ABB RAPID module: TaskModule.mod

MODULE TaskModule
    !*****************************************************
    !Module Name: TaskModule
    !Version:     1.0
    !Description: This module stroes ths data which are not shared among other tasks
    !Date:        2018-8-10
    !Author:      Michael
    !*****************************************************

    VAR num numStation:=1;
    VAR partdata pdTmpChk;
    VAR string sPartDataName;

    VAR syncident SyncPositionerHomed;
    VAR syncident SyncWobjScanning;
    VAR syncident SyncWobjBranchScaning;
    VAR syncident SyncWobjBranchScaned;
    VAR syncident SyncWobjHeaderScaning;
    VAR syncident SyncWobjHeaderScaned;
    VAR syncident SyncWobjBranchScaningV2;
    VAR syncident SyncWobjBranchScanedV2;
    VAR syncident SyncWobjHeaderScaningV2;
    VAR syncident SyncWobjHeaderScanedV2;
    VAR syncident SyncBranchPeripherySmarTac;
    VAR syncident SyncHeaderPeripherySmarTac;
    VAR syncident SyncWobjScaned;
    VAR syncident SyncWobjRevised;

    VAR syncident SyncPositionerWeldApproached;
    VAR syncident SyncRobotsWeldApproached;
    VAR syncident SyncAllRobotsWeldStart;
    VAR syncident SyncAllRobotsWeldEnd;
    VAR syncident SyncRobotsWeldDeparted;

    VAR syncident SyncMoveLSubstituted1;
    VAR syncident SyncMoveLSubstituted2;

    VAR syncident SyncRobotsForTest11;
    VAR syncident SyncRobotsForTest12;
    VAR syncident SyncRobotsForTest13;

    VAR syncident SyncRobotsForTest21;
    VAR syncident SyncRobotsForTest22;
    VAR syncident SyncRobotsForTest23;
    VAR syncident SyncRobotsForTest24;
    VAR syncident SyncRobotsForTest25;
    VAR syncident SyncRobotsForTest26;

    VAR syncident SyncVerifyTrackHorizontal1;
    VAR syncident SyncVerifyTrackHorizontal2;
    VAR syncident SyncVerifyTrackHorizontal3;
    VAR syncident SyncVerifyTrackHorizontal4;
    VAR syncident SyncVerifyTrackHorizontal5;
    VAR syncident SyncVerifyTrackHorizontal6;
    VAR syncident SyncVerifyTrackHorizontal7;
    VAR syncident SyncVerifyTrackHorizontal8;

    VAR string strCurTaskName:="T_ROB2";
    VAR num numCurTaskNo:=2;
    VAR num numRobLayerCurTotal;
    VAR RECORDWeldTarget rRobLayerCur{30};

    TASK PERS tooldata toolWeldGun:=[TRUE,[[79.6797,-0.416093,372.923],[0.951182,0.000468257,0.308629,0.000774227]],[5.2,[30.6,-22.1,100.1],[1,0,0,0],0,0,0]];
    TASK PERS tooldata toolLaser:=[TRUE,[[-50.2332,13.2462,422.412],[0.99997,-0.00371251,-0.00510598,-0.00440267]],[5.2,[30.6,-22.1,100.1],[1,0,0,0],0,0,0]];
    TASK PERS extjoint extjointValue:=[3962.74,9E+09,9E+09,9E+09,9E+09,9E+09];

    TASK PERS robtarget robtApproachPlatoonSinking:=[[380,200,190.09],[0.24541,0.749,0.614742,-0.0294245],[-1,-1,0,1],[4837,9E+09,9E+09,9E+09,9E+09,9E+09]];
    TASK PERS robtarget robtDepartPlatoonSinking:=[[380,200,190.09],[0.245412,0.748999,0.614742,-0.0294268],[-1,-1,0,1],[4837,9E+09,9E+09,9E+09,9E+09,9E+09]];

    TASK PERS robtarget robtApproachSaddle:=[[487.15,620.91,295.61],[0.42303,-0.434139,-0.767759,0.207644],[0,-1,0,0],[4837,9E+09,9E+09,9E+09,9E+09,9E+09]];
    TASK PERS robtarget robtDepartSaddle:=[[487.15,238.1,333.7],[0.270598,0.653282,-0.653281,0.270598],[0,-1,-2,0],[4837,9E+09,9E+09,9E+09,9E+09,9E+09]];

    TASK PERS robtarget robtApproachSaddleScan:=[[380,426.46,263.71],[0.0219383,0.0029599,-0.868719,0.494811],[-1,-1,-1,1],[4837,9E+09,9E+09,9E+09,9E+09,9E+09]];
    TASK PERS robtarget robtDepartSaddleScan:=[[380,426.46,263.71],[0.0219385,0.00296103,-0.868717,0.494814],[-1,-1,-1,1],[4837,9E+09,9E+09,9E+09,9E+09,9E+09]];

    TASK PERS robtarget robtApproachPlatoonSinkingScan:=[[380,238.1,333.7],[0.270598,0.653281,-0.653282,0.270598],[0,0,1,1],[4837,9E+09,9E+09,9E+09,9E+09,9E+09]];
    TASK PERS robtarget robtDepartPlatoonSinkingScan:=[[380,238.1,333.7],[0.270598,0.653281,-0.653282,0.270598],[0,0,1,1],[4837,9E+09,9E+09,9E+09,9E+09,9E+09]];

    TASK PERS confdata confPlatoonSinkingOrigin:=[0,0,0,1];
    TASK PERS confdata confSaddleOrigin:=[0,-1,0,0];

    TASK PERS robtarget robtNext:=[[39.1752,-5.3,137.55],[0.0379422,0.543848,0.68392,-0.484813],[0,0,-1,1],[447,9E+09,9E+09,9E+09,9E+09,9E+09]];
    TASK PERS robtarget robtCircleEnd:=[[37.5661,-7.30249,138.697],[0.0379422,0.543848,0.68392,-0.484813],[-1,-1,-1,1],[2602,9E+09,9E+09,9E+09,9E+09,9E+09]];

    TASK PERS seamdata seamNext:=[0,0.5,[0,0,0,100,0,0,0,0,0],0,0,5,0,0,[0,0,1,140,0,0,0,0,0],0,1.5,[0,0,1,90,0,0,0,0,0],0.04,0,[0,0,0,0,0,0,0,0,0],0.5];
    TASK PERS welddata weldNext:=[7,0,[25,0,0,0,0,200,0,0,0],[0,0,0,0,0,0,0,0,0]];
    TASK PERS weavedata weaveNext:=[0,0,0,0,0,0,0,0,0,0,0,0,0,0,0];
    TASK PERS trackdata trackNext:=[0,FALSE,50,[0,0,0,0,0,0,0,0,0],[0,0,0,0,0,0,0]];
    TASK PERS adaptdata adaptNext:=[0,1,0,0,0.1,100,0.1,100];
    TASK PERS num numWeaveWidth90:=0;
    TASK PERS num numGrooveWidthNext:=0.1;

    TASK PERS jointtarget jointNext:=[[9E+09,9E+09,9E+09,9E+09,9E+09,9E+09],[0,66.4272,9E+09,9E+09,9E+09,9E+09]];

    VAR clock clockPartTimeConsume;
    TASK PERS num numTimeConsumeTotal:=683.013;

    CONST string strWeldProcedureLogLogFileName:="WeldProcedureLog2.csv";

    CONST string strSSBLogFileName:="ScanSaddleBranch2.csv";
    CONST string strSSHLogFileName:="ScanSaddleHeader2.csv";

    !For branch SmarTac
    TASK PERS num numSSBPointsTotal:=13;
    !Scan branch range
    TASK PERS num numSSBAngleFrom:=125;
    TASK PERS num numSSBAngleTo:=30;

    !For saddle header SmarTac
    TASK PERS num numSSHPointsTotal:=13;
    !Scan saddle header range
    TASK PERS num numSSHAngleFrom:=0;
    TASK PERS num numSSHAngleTo:=90;

    !Scan saddle branch points
    TASK PERS robtarget robtSSBLaserSmarTacs{20}:=[[[923.658,130.45,259.25],[0.67438,0.67438,0.212631,0.212631],[-1,-1,1,1],[4202,9E+09,9E+09,9E+09,9E+09,9E+09]],[[942.496,141.787,259.25],[0.687449,0.687449,0.165571,0.165571],[-1,-1,1,1],[4202,9E+09,9E+09,9E+09,9E+09,9E+09]],[[962.716,150.422,259.25],[0.697239,0.697239,0.11772,0.11772],[-1,-1,1,1],[4202,9E+09,9E+09,9E+09,9E+09,9E+09]],[[983.932,156.19,259.25],[0.703702,0.703702,0.0693086,0.0693086],[-1,-1,1,1],[4202,9E+09,9E+09,9E+09,9E+09,9E+09]],[[1005.74,158.981,259.25],[0.706808,0.706808,0.020566,0.020566],[-1,-1,1,1],[4202,9E+09,9E+09,9E+09,9E+09,9E+09]],[[1027.73,158.741,259.25],[0.706541,0.706541,-0.0282747,-0.0282747],[0,0,1,1],[4202,9E+09,9E+09,9E+09,9E+09,9E+09]],[[1049.47,155.475,259.25],[0.702904,0.702904,-0.0769805,-0.0769805],[0,0,0,1],[4202,9E+09,9E+09,9E+09,9E+09,9E+09]],[[1070.55,149.246,259.25],[0.695913,0.695913,-0.125319,-0.125319],[0,0,0,1],[4202,9E+09,9E+09,9E+09,9E+09,9E+09]],[[1090.58,140.172,259.25],[0.685602,0.685602,-0.17306,-0.17306],[0,0,0,1],[4202,9E+09,9E+09,9E+09,9E+09,9E+09]],[[1109.17,128.426,259.25],[0.67202,0.67202,-0.219975,-0.219975],[0,0,0,1],[4202,9E+09,9E+09,9E+09,9E+09,9E+09]],[[1125.96,114.233,259.25],[0.655232,0.655232,-0.26584,-0.26584],[0,0,0,1],[4202,9E+09,9E+09,9E+09,9E+09,9E+09]],[[1140.63,97.8615,259.25],[0.635318,0.635318,-0.310437,-0.310437],[0,0,0,1],[4202,9E+09,9E+09,9E+09,9E+09,9E+09]],[[1152.91,79.625,259.25],[0.612372,0.612372,-0.353553,-0.353553],[0,0,0,1],[4202,9E+09,9E+09,9E+09,9E+09,9E+09]],[[652.53,-493.33,1047.99],[0.459259,-0.544323,-0.447932,-0.54051],[0,0,0,1],[4837,9E+09,9E+09,9E+09,9E+09,9E+09]],[[652.53,-493.33,1047.99],[0.459259,-0.544323,-0.447932,-0.54051],[-1,0,-2,1],[4837,9E+09,9E+09,9E+09,9E+09,9E+09]],[[652.53,-493.33,1047.99],[0.459259,-0.544323,-0.447932,-0.54051],[-1,0,-2,1],[4837,9E+09,9E+09,9E+09,9E+09,9E+09]],[[652.53,-493.33,1047.99],[0.459259,-0.544323,-0.447932,-0.54051],[-1,0,-2,1],[4837,9E+09,9E+09,9E+09,9E+09,9E+09]],[[652.53,-493.33,1047.99],[0.459259,-0.544323,-0.447932,-0.54051],[-1,0,-2,1],[4837,9E+09,9E+09,9E+09,9E+09,9E+09]],[[652.53,-493.33,1047.99],[0.459259,-0.544323,-0.447932,-0.54051],[-1,0,-2,1],[4837,9E+09,9E+09,9E+09,9E+09,9E+09]],[[652.53,-493.33,1047.99],[0.459259,-0.544323,-0.447932,-0.54051],[-1,0,-2,1],[4837,9E+09,9E+09,9E+09,9E+09,9E+09]]];
    TASK PERS robtarget robtSSBWireSmarTacs{20}:=[[[428.493,28.575,188.15],[0.683013,0.183013,-0.683013,0.183013],[0,1,-3,1],[4838,9E+09,9E+09,9E+09,9E+09,9E+09]],[[422.779,36.7353,188.15],[0.664463,0.241845,-0.664463,0.241845],[0,1,-3,1],[4838,9E+09,9E+09,9E+09,9E+09,9E+09]],[[415.735,43.7794,188.15],[0.640856,0.298836,-0.640856,0.298836],[0,1,-3,1],[4838,9E+09,9E+09,9E+09,9E+09,9E+09]],[[407.575,49.4934,188.15],[0.612372,0.353553,-0.612372,0.353553],[0,0,-3,1],[4838,9E+09,9E+09,9E+09,9E+09,9E+09]],[[398.546,53.7034,188.15],[0.579228,0.40558,-0.579228,0.40558],[0,0,-3,1],[4838,9E+09,9E+09,9E+09,9E+09,9E+09]],[[388.924,56.2818,188.15],[0.541675,0.454519,-0.541675,0.454519],[0,0,-3,1],[4838,9E+09,9E+09,9E+09,9E+09,9E+09]],[[379,57.15,188.15],[0.5,0.5,-0.5,0.5],[0,0,-3,1],[4838,9E+09,9E+09,9E+09,9E+09,9E+09]],[[369.076,56.2818,188.15],[0.454519,0.541675,-0.454519,0.541675],[-1,-1,-2,1],[4838,9E+09,9E+09,9E+09,9E+09,9E+09]],[[359.454,53.7034,188.15],[0.40558,0.579228,-0.40558,0.579228],[-1,-1,-2,1],[4838,9E+09,9E+09,9E+09,9E+09,9E+09]],[[350.425,49.4934,188.15],[0.353553,0.612372,-0.353553,0.612372],[-1,-1,-2,1],[4838,9E+09,9E+09,9E+09,9E+09,9E+09]],[[342.265,43.7794,188.15],[0.298836,0.640856,-0.298836,0.640856],[-1,-2,-2,1],[4838,9E+09,9E+09,9E+09,9E+09,9E+09]],[[335.221,36.7353,188.15],[0.241845,0.664463,-0.241845,0.664463],[-1,-2,-2,1],[4838,9E+09,9E+09,9E+09,9E+09,9E+09]],[[329.507,28.575,188.15],[0.183013,0.683013,-0.183013,0.683013],[-1,-2,-2,1],[4838,9E+09,9E+09,9E+09,9E+09,9E+09]],[[652.53,-493.33,1047.99],[0.459259,-0.544323,-0.447932,-0.54051],[-1,-1,-2,1],[4837,9E+09,9E+09,9E+09,9E+09,9E+09]],[[652.53,-493.33,1047.99],[0.459259,-0.544323,-0.447932,-0.54051],[-1,0,-2,1],[4837,9E+09,9E+09,9E+09,9E+09,9E+09]],[[652.53,-493.33,1047.99],[0.459259,-0.544323,-0.447932,-0.54051],[-1,0,-2,1],[4837,9E+09,9E+09,9E+09,9E+09,9E+09]],[[652.53,-493.33,1047.99],[0.459259,-0.544323,-0.447932,-0.54051],[-1,0,-2,1],[4837,9E+09,9E+09,9E+09,9E+09,9E+09]],[[652.53,-493.33,1047.99],[0.459259,-0.544323,-0.447932,-0.54051],[-1,0,-2,1],[4837,9E+09,9E+09,9E+09,9E+09,9E+09]],[[652.53,-493.33,1047.99],[0.459259,-0.544323,-0.447932,-0.54051],[-1,0,-2,1],[4837,9E+09,9E+09,9E+09,9E+09,9E+09]],[[652.53,-493.33,1047.99],[0.459259,-0.544323,-0.447932,-0.54051],[-1,0,-2,1],[4837,9E+09,9E+09,9E+09,9E+09,9E+09]]];
    TASK PERS robtarget robtSSBLinerFrom:=[[427.815,90,259.25],[0.707107,0.707107,0,0],[0,0,1,1],[4202,9E+09,9E+09,9E+09,9E+09,9E+09]];
    TASK PERS robtarget robtSSBLinerTo:=[[427.815,90,259.25],[0.707107,0.707107,0,0],[0,0,1,1],[4202,9E+09,9E+09,9E+09,9E+09,9E+09]];

    !Scan saddle branch results, shared for all the four scan methods
    TASK PERS pose poseSSBs{20}:=[[[-1.32358,1.90598,0.00161743],[1,0,0,0]],[[-0.951538,1.84398,-0.0424805],[1,0,0,0]],[[-0.775452,2.22177,-0.0251465],[1,0,0,0]],[[-0.413208,2.22758,0.000427246],[1,0,0,0]],[[-0.156219,2.60087,-0.0246429],[1,0,0,0]],[[0.213074,2.58353,0.020462],[1,0,0,0]],[[0.449005,2.08419,-0.0298309],[1,0,0,0]],[[0.743073,1.96958,-0.0420227],[1,0,0,0]],[[1.15472,2.18119,0.0494232],[1,0,0,0]],[[1.04321,1.4268,-0.00532532],[1,0,0,0]],[[1.86594,1.89365,0.0466766],[1,0,0,0]],[[1.22217,0.918324,-0.00390625],[1,0,0,0]],[[0.608215,0.37476,-0.00968933],[1,0,0,0]],[[0,0,0],[1,0,0,0]],[[0,0,0],[1,0,0,0]],[[0,0,0],[1,0,0,0]],[[0,0,0],[1,0,0,0]],[[0,0,0],[1,0,0,0]],[[0,0,0],[1,0,0,0]],[[0,0,0],[1,0,0,0]]];
    TASK PERS num numSSBLaserValues{100}:=[0,0,0,0,0,0,0,0,0,0,0,0,0,0,0,0,0,0,0,0,0,0,0,0,0,0,0,0,0,0,0,0,0,0,0,0,0,0,0,0,0,0,0,0,0,0,0,0,0,0,0,0,0,0,0,0,0,0,0,0,0,0,0,0,0,0,0,0,0,0,0,0,0,0,0,0,0,0,0,0,0,0,0,0,0,0,0,0,0,0,0,0,0,0,0,0,0,0,0,0];
    TASK PERS robtarget robtSSBPeripherys{100}:=[[[345.897,48.7205,208.152],[0.674376,0.674381,0.212635,0.212635],[-1,-1,1,1],[4837,9E+09,9E+09,9E+09,9E+09,9E+09]],[[353.029,52.7272,208.108],[0.687429,0.687473,0.165559,0.165568],[-1,-1,1,1],[4837,9E+09,9E+09,9E+09,9E+09,9E+09]],[[360.461,56.2038,208.125],[0.697234,0.697245,0.117717,0.11772],[-1,-1,1,1],[4837,9E+09,9E+09,9E+09,9E+09,9E+09]],[[368.437,58.2795,208.15],[0.703708,0.703694,0.0693283,0.0693077],[-1,-1,1,1],[4837,9E+09,9E+09,9E+09,9E+09,9E+09]],[[376.521,59.6542,208.125],[0.706794,0.706822,0.0205642,0.0205642],[-1,-1,1,1],[4837,9E+09,9E+09,9E+09,9E+09,9E+09]],[[384.78,59.5508,208.17],[0.706548,0.706534,-0.0282861,-0.0282663],[0,0,0,1],[4837,9E+09,9E+09,9E+09,9E+09,9E+09]],[[392.819,57.8795,208.12],[0.702889,0.702918,-0.0769979,-0.0769742],[0,0,0,1],[4836.99,9E+09,9E+09,9E+09,9E+09,9E+09]],[[400.68,55.5295,208.108],[0.695903,0.695926,-0.125326,-0.125296],[0,0,0,1],[4837,9E+09,9E+09,9E+09,9E+09,9E+09]],[[408.278,52.4847,208.199],[0.685623,0.685578,-0.173065,-0.173068],[0,0,0,1],[4837,9E+09,9E+09,9E+09,9E+09,9E+09]],[[414.837,47.5151,208.145],[0.672022,0.672019,-0.219953,-0.219993],[0,0,0,1],[4837,9E+09,9E+09,9E+09,9E+09,9E+09]],[[421.685,42.8883,208.197],[0.655247,0.655221,-0.265826,-0.265844],[0,0,0,1],[4837,9E+09,9E+09,9E+09,9E+09,9E+09]],[[426.308,36.0378,208.146],[0.635315,0.635323,-0.310461,-0.310408],[0,0,0,1],[4837,9E+09,9E+09,9E+09,9E+09,9E+09]],[[430.102,28.9498,208.14],[0.612373,0.612366,-0.353539,-0.353577],[0,0,0,1],[4837,9E+09,9E+09,9E+09,9E+09,9E+09]],[[75.54,-110.49,75.53],[0.104911,-0.592891,0.59209,0.535634],[-1,-2,0,1],[3747.5,9E+09,9E+09,9E+09,9E+09,9E+09]],[[75.54,-110.49,75.53],[0.104911,-0.592891,0.59209,0.535634],[-1,0,-1,0],[3747.5,9E+09,9E+09,9E+09,9E+09,9E+09]],[[75.54,-110.49,75.53],[0.104911,-0.592891,0.59209,0.535634],[-1,0,-1,0],[3747.5,9E+09,9E+09,9E+09,9E+09,9E+09]],[[75.54,-110.49,75.53],[0.104911,-0.592891,0.59209,0.535634],[-1,0,-1,0],[3747.5,9E+09,9E+09,9E+09,9E+09,9E+09]],[[75.54,-110.49,75.53],[0.104911,-0.592891,0.59209,0.535634],[-1,0,-1,0],[3747.5,9E+09,9E+09,9E+09,9E+09,9E+09]],[[75.54,-110.49,75.53],[0.104911,-0.592891,0.59209,0.535634],[-1,0,-1,0],[3747.5,9E+09,9E+09,9E+09,9E+09,9E+09]],[[75.54,-110.49,75.53],[0.104911,-0.592891,0.59209,0.535634],[-1,0,-1,0],[3747.5,9E+09,9E+09,9E+09,9E+09,9E+09]],[[75.54,-110.49,75.53],[0.104911,-0.592891,0.59209,0.535634],[-1,0,-1,0],[3747.5,9E+09,9E+09,9E+09,9E+09,9E+09]],[[75.54,-110.49,75.53],[0.104911,-0.592891,0.59209,0.535634],[-1,0,-1,0],[3747.5,9E+09,9E+09,9E+09,9E+09,9E+09]],[[75.54,-110.49,75.53],[0.104911,-0.592891,0.59209,0.535634],[-1,0,-1,0],[3747.5,9E+09,9E+09,9E+09,9E+09,9E+09]],[[75.54,-110.49,75.53],[0.104911,-0.592891,0.59209,0.535634],[-1,0,-1,0],[3747.5,9E+09,9E+09,9E+09,9E+09,9E+09]],[[75.54,-110.49,75.53],[0.104911,-0.592891,0.59209,0.535634],[-1,0,-1,0],[3747.5,9E+09,9E+09,9E+09,9E+09,9E+09]],[[75.54,-110.49,75.53],[0.104911,-0.592891,0.59209,0.535634],[-1,0,-1,0],[3747.5,9E+09,9E+09,9E+09,9E+09,9E+09]],[[75.54,-110.49,75.53],[0.104911,-0.592891,0.59209,0.535634],[-1,0,-1,0],[3747.5,9E+09,9E+09,9E+09,9E+09,9E+09]],[[75.54,-110.49,75.53],[0.104911,-0.592891,0.59209,0.535634],[-1,0,-1,0],[3747.5,9E+09,9E+09,9E+09,9E+09,9E+09]],[[75.54,-110.49,75.53],[0.104911,-0.592891,0.59209,0.535634],[-1,0,-1,0],[3747.5,9E+09,9E+09,9E+09,9E+09,9E+09]],[[75.54,-110.49,75.53],[0.104911,-0.592891,0.59209,0.535634],[-1,0,-1,0],[3747.5,9E+09,9E+09,9E+09,9E+09,9E+09]],[[75.54,-110.49,75.53],[0.104911,-0.592891,0.59209,0.535634],[-1,0,-1,0],[3747.5,9E+09,9E+09,9E+09,9E+09,9E+09]],[[75.54,-110.49,75.53],[0.104911,-0.592891,0.59209,0.535634],[-1,0,-1,0],[3747.5,9E+09,9E+09,9E+09,9E+09,9E+09]],[[75.54,-110.49,75.53],[0.104911,-0.592891,0.59209,0.535634],[-1,0,-1,0],[3747.5,9E+09,9E+09,9E+09,9E+09,9E+09]],[[75.54,-110.49,75.53],[0.104911,-0.592891,0.59209,0.535634],[-1,0,-1,0],[3747.5,9E+09,9E+09,9E+09,9E+09,9E+09]],[[75.54,-110.49,75.53],[0.104911,-0.592891,0.59209,0.535634],[-1,0,-1,0],[3747.5,9E+09,9E+09,9E+09,9E+09,9E+09]],[[75.54,-110.49,75.53],[0.104911,-0.592891,0.59209,0.535634],[-1,0,-1,0],[3747.5,9E+09,9E+09,9E+09,9E+09,9E+09]],[[75.54,-110.49,75.53],[0.104911,-0.592891,0.59209,0.535634],[-1,0,-1,0],[3747.5,9E+09,9E+09,9E+09,9E+09,9E+09]],[[75.54,-110.49,75.53],[0.104911,-0.592891,0.59209,0.535634],[-1,0,-1,0],[3747.5,9E+09,9E+09,9E+09,9E+09,9E+09]],[[75.54,-110.49,75.53],[0.104911,-0.592891,0.59209,0.535634],[-1,0,-1,0],[3747.5,9E+09,9E+09,9E+09,9E+09,9E+09]],[[75.54,-110.49,75.53],[0.104911,-0.592891,0.59209,0.535634],[-1,0,-1,0],[3747.5,9E+09,9E+09,9E+09,9E+09,9E+09]],[[75.54,-110.49,75.53],[0.104911,-0.592891,0.59209,0.535634],[-1,0,-1,0],[3747.5,9E+09,9E+09,9E+09,9E+09,9E+09]],[[75.54,-110.49,75.53],[0.104911,-0.592891,0.59209,0.535634],[-1,0,-1,0],[3747.5,9E+09,9E+09,9E+09,9E+09,9E+09]],[[75.54,-110.49,75.53],[0.104911,-0.592891,0.59209,0.535634],[-1,0,-1,0],[3747.5,9E+09,9E+09,9E+09,9E+09,9E+09]],[[75.54,-110.49,75.53],[0.104911,-0.592891,0.59209,0.535634],[-1,0,-1,0],[3747.5,9E+09,9E+09,9E+09,9E+09,9E+09]],[[75.54,-110.49,75.53],[0.104911,-0.592891,0.59209,0.535634],[-1,0,-1,0],[3747.5,9E+09,9E+09,9E+09,9E+09,9E+09]],[[75.54,-110.49,75.53],[0.104911,-0.592891,0.59209,0.535634],[-1,0,-1,0],[3747.5,9E+09,9E+09,9E+09,9E+09,9E+09]],[[75.54,-110.49,75.53],[0.104911,-0.592891,0.59209,0.535634],[-1,0,-1,0],[3747.5,9E+09,9E+09,9E+09,9E+09,9E+09]],[[75.54,-110.49,75.53],[0.104911,-0.592891,0.59209,0.535634],[-1,0,-1,0],[3747.5,9E+09,9E+09,9E+09,9E+09,9E+09]],[[75.54,-110.49,75.53],[0.104911,-0.592891,0.59209,0.535634],[-1,0,-1,0],[3747.5,9E+09,9E+09,9E+09,9E+09,9E+09]],[[75.54,-110.49,75.53],[0.104911,-0.592891,0.59209,0.535634],[-1,0,-1,0],[3747.5,9E+09,9E+09,9E+09,9E+09,9E+09]],[[75.54,-110.49,75.53],[0.104911,-0.592891,0.59209,0.535634],[-1,0,-1,0],[3747.5,9E+09,9E+09,9E+09,9E+09,9E+09]],[[75.54,-110.49,75.53],[0.104911,-0.592891,0.59209,0.535634],[-1,0,-1,0],[3747.5,9E+09,9E+09,9E+09,9E+09,9E+09]],[[75.54,-110.49,75.53],[0.104911,-0.592891,0.59209,0.535634],[-1,0,-1,0],[3747.5,9E+09,9E+09,9E+09,9E+09,9E+09]],[[75.54,-110.49,75.53],[0.104911,-0.592891,0.59209,0.535634],[-1,0,-1,0],[3747.5,9E+09,9E+09,9E+09,9E+09,9E+09]],[[75.54,-110.49,75.53],[0.104911,-0.592891,0.59209,0.535634],[-1,0,-1,0],[3747.5,9E+09,9E+09,9E+09,9E+09,9E+09]],[[75.54,-110.49,75.53],[0.104911,-0.592891,0.59209,0.535634],[-1,0,-1,0],[3747.5,9E+09,9E+09,9E+09,9E+09,9E+09]],[[75.54,-110.49,75.53],[0.104911,-0.592891,0.59209,0.535634],[-1,0,-1,0],[3747.5,9E+09,9E+09,9E+09,9E+09,9E+09]],[[75.54,-110.49,75.53],[0.104911,-0.592891,0.59209,0.535634],[-1,0,-1,0],[3747.5,9E+09,9E+09,9E+09,9E+09,9E+09]],[[75.54,-110.49,75.53],[0.104911,-0.592891,0.59209,0.535634],[-1,0,-1,0],[3747.5,9E+09,9E+09,9E+09,9E+09,9E+09]],[[75.54,-110.49,75.53],[0.104911,-0.592891,0.59209,0.535634],[-1,0,-1,0],[3747.5,9E+09,9E+09,9E+09,9E+09,9E+09]],[[75.54,-110.49,75.53],[0.104911,-0.592891,0.59209,0.535634],[-1,0,-1,0],[3747.5,9E+09,9E+09,9E+09,9E+09,9E+09]],[[75.54,-110.49,75.53],[0.104911,-0.592891,0.59209,0.535634],[-1,0,-1,0],[3747.5,9E+09,9E+09,9E+09,9E+09,9E+09]],[[75.54,-110.49,75.53],[0.104911,-0.592891,0.59209,0.535634],[-1,0,-1,0],[3747.5,9E+09,9E+09,9E+09,9E+09,9E+09]],[[75.54,-110.49,75.53],[0.104911,-0.592891,0.59209,0.535634],[-1,0,-1,0],[3747.5,9E+09,9E+09,9E+09,9E+09,9E+09]],[[75.54,-110.49,75.53],[0.104911,-0.592891,0.59209,0.535634],[-1,0,-1,0],[3747.5,9E+09,9E+09,9E+09,9E+09,9E+09]],[[75.54,-110.49,75.53],[0.104911,-0.592891,0.59209,0.535634],[-1,0,-1,0],[3747.5,9E+09,9E+09,9E+09,9E+09,9E+09]],[[75.54,-110.49,75.53],[0.104911,-0.592891,0.59209,0.535634],[-1,0,-1,0],[3747.5,9E+09,9E+09,9E+09,9E+09,9E+09]],[[75.54,-110.49,75.53],[0.104911,-0.592891,0.59209,0.535634],[-1,0,-1,0],[3747.5,9E+09,9E+09,9E+09,9E+09,9E+09]],[[75.54,-110.49,75.53],[0.104911,-0.592891,0.59209,0.535634],[-1,0,-1,0],[3747.5,9E+09,9E+09,9E+09,9E+09,9E+09]],[[75.54,-110.49,75.53],[0.104911,-0.592891,0.59209,0.535634],[-1,0,-1,0],[3747.5,9E+09,9E+09,9E+09,9E+09,9E+09]],[[75.54,-110.49,75.53],[0.104911,-0.592891,0.59209,0.535634],[-1,0,-1,0],[3747.5,9E+09,9E+09,9E+09,9E+09,9E+09]],[[75.54,-110.49,75.53],[0.104911,-0.592891,0.59209,0.535634],[-1,0,-1,0],[3747.5,9E+09,9E+09,9E+09,9E+09,9E+09]],[[75.54,-110.49,75.53],[0.104911,-0.592891,0.59209,0.535634],[-1,0,-1,0],[3747.5,9E+09,9E+09,9E+09,9E+09,9E+09]],[[75.54,-110.49,75.53],[0.104911,-0.592891,0.59209,0.535634],[-1,0,-1,0],[3747.5,9E+09,9E+09,9E+09,9E+09,9E+09]],[[75.54,-110.49,75.53],[0.104911,-0.592891,0.59209,0.535634],[-1,0,-1,0],[3747.5,9E+09,9E+09,9E+09,9E+09,9E+09]],[[75.54,-110.49,75.53],[0.104911,-0.592891,0.59209,0.535634],[-1,0,-1,0],[3747.5,9E+09,9E+09,9E+09,9E+09,9E+09]],[[75.54,-110.49,75.53],[0.104911,-0.592891,0.59209,0.535634],[-1,0,-1,0],[3747.5,9E+09,9E+09,9E+09,9E+09,9E+09]],[[75.54,-110.49,75.53],[0.104911,-0.592891,0.59209,0.535634],[-1,0,-1,0],[3747.5,9E+09,9E+09,9E+09,9E+09,9E+09]],[[75.54,-110.49,75.53],[0.104911,-0.592891,0.59209,0.535634],[-1,0,-1,0],[3747.5,9E+09,9E+09,9E+09,9E+09,9E+09]],[[75.54,-110.49,75.53],[0.104911,-0.592891,0.59209,0.535634],[-1,0,-1,0],[3747.5,9E+09,9E+09,9E+09,9E+09,9E+09]],[[75.54,-110.49,75.53],[0.104911,-0.592891,0.59209,0.535634],[-1,0,-1,0],[3747.5,9E+09,9E+09,9E+09,9E+09,9E+09]],[[75.54,-110.49,75.53],[0.104911,-0.592891,0.59209,0.535634],[-1,0,-1,0],[3747.5,9E+09,9E+09,9E+09,9E+09,9E+09]],[[75.54,-110.49,75.53],[0.104911,-0.592891,0.59209,0.535634],[-1,0,-1,0],[3747.5,9E+09,9E+09,9E+09,9E+09,9E+09]],[[75.54,-110.49,75.53],[0.104911,-0.592891,0.59209,0.535634],[-1,0,-1,0],[3747.5,9E+09,9E+09,9E+09,9E+09,9E+09]],[[75.54,-110.49,75.53],[0.104911,-0.592891,0.59209,0.535634],[-1,0,-1,0],[3747.5,9E+09,9E+09,9E+09,9E+09,9E+09]],[[75.54,-110.49,75.53],[0.104911,-0.592891,0.59209,0.535634],[-1,0,-1,0],[3747.5,9E+09,9E+09,9E+09,9E+09,9E+09]],[[75.54,-110.49,75.53],[0.104911,-0.592891,0.59209,0.535634],[-1,0,-1,0],[3747.5,9E+09,9E+09,9E+09,9E+09,9E+09]],[[75.54,-110.49,75.53],[0.104911,-0.592891,0.59209,0.535634],[-1,0,-1,0],[3747.5,9E+09,9E+09,9E+09,9E+09,9E+09]],[[75.54,-110.49,75.53],[0.104911,-0.592891,0.59209,0.535634],[-1,0,-1,0],[3747.5,9E+09,9E+09,9E+09,9E+09,9E+09]],[[75.54,-110.49,75.53],[0.104911,-0.592891,0.59209,0.535634],[-1,0,-1,0],[3747.5,9E+09,9E+09,9E+09,9E+09,9E+09]],[[75.54,-110.49,75.53],[0.104911,-0.592891,0.59209,0.535634],[-1,0,-1,0],[3747.5,9E+09,9E+09,9E+09,9E+09,9E+09]],[[75.54,-110.49,75.53],[0.104911,-0.592891,0.59209,0.535634],[-1,0,-1,0],[3747.5,9E+09,9E+09,9E+09,9E+09,9E+09]],[[75.54,-110.49,75.53],[0.104911,-0.592891,0.59209,0.535634],[-1,0,-1,0],[3747.5,9E+09,9E+09,9E+09,9E+09,9E+09]],[[75.54,-110.49,75.53],[0.104911,-0.592891,0.59209,0.535634],[-1,0,-1,0],[3747.5,9E+09,9E+09,9E+09,9E+09,9E+09]],[[75.54,-110.49,75.53],[0.104911,-0.592891,0.59209,0.535634],[-1,0,-1,0],[3747.5,9E+09,9E+09,9E+09,9E+09,9E+09]],[[75.54,-110.49,75.53],[0.104911,-0.592891,0.59209,0.535634],[-1,0,-1,0],[3747.5,9E+09,9E+09,9E+09,9E+09,9E+09]],[[75.54,-110.49,75.53],[0.104911,-0.592891,0.59209,0.535634],[-1,0,-1,0],[3747.5,9E+09,9E+09,9E+09,9E+09,9E+09]],[[75.54,-110.49,75.53],[0.104911,-0.592891,0.59209,0.535634],[-1,0,-1,0],[3747.5,9E+09,9E+09,9E+09,9E+09,9E+09]],[[75.54,-110.49,75.53],[0.104911,-0.592891,0.59209,0.535634],[-1,0,-1,0],[3747.5,9E+09,9E+09,9E+09,9E+09,9E+09]],[[75.54,-110.49,75.53],[0.104911,-0.592891,0.59209,0.535634],[-1,0,-1,0],[3747.5,9E+09,9E+09,9E+09,9E+09,9E+09]]];
    TASK PERS pos posSSBPeripherys{100}:=[[345.897,48.7205,208.152],[353.029,52.7272,208.108],[360.461,56.2038,208.125],[368.437,58.2795,208.15],[376.521,59.6542,208.125],[384.78,59.5508,208.17],[392.819,57.8795,208.12],[400.68,55.5295,208.108],[408.278,52.4847,208.199],[414.837,47.5151,208.145],[421.685,42.8883,208.197],[426.308,36.0378,208.146],[430.102,28.9498,208.14],[403.721,-54.5007,218.144],[402.695,-54.7914,218.15],[401.613,-55.2287,218.151],[400.612,-55.6663,218.16],[399.584,-55.6652,218.161],[398.506,-55.6653,218.154],[397.454,-56.5454,218.153],[396.435,-56.5484,218.147],[395.393,-57.1338,218.149],[394.377,-57.573,218.149],[393.302,-57.5728,218.152],[392.269,-57.8653,218.151],[391.229,-58.0135,218.151],[390.146,-58.0121,218.15],[389.116,-58.1615,218.148],[388.11,-58.601,218.152],[387.028,-58.5999,218.152],[386,-58.6,218.154],[384.982,-58.6014,218.153],[383.916,-58.4571,218.152],[382.868,-58.6069,218.153],[381.835,-58.4659,218.153],[380.789,-58.1789,218.151],[379.733,-58.1848,218.151],[378.699,-58.6326,218.147],[377.665,-58.489,218.152],[376.646,-58.486,218.161],[375.577,-58.6304,218.172],[374.516,-57.3071,218.178],[373.483,-57.5924,218.186],[372.468,-58.4606,218.198],[371.413,-56.8386,218.212],[370.378,-57.1252,218.221],[369.332,-56.8308,218.22],[368.287,-57.1221,218.223],[367.205,-56.5413,218.213],[366.179,-55.6646,218.209],[365.152,-55.668,218.196],[364.087,-55.0838,218.188],[363.017,-55.232,218.18],[361.985,-54.7921,218.174],[360.946,-54.4989,218.172],[359.89,-53.7688,218.165],[358.836,-54.0598,218.167],[357.811,-53.3263,218.165],[356.755,-52.301,218.162],[355.671,-51.7184,218.156],[354.682,-51.1319,218.154],[353.654,-50.5491,218.148],[352.593,-50.4035,218.147],[351.534,-50.1095,218.146],[350.499,-49.3779,218.145],[349.454,-48.3511,218.147],[348.381,-47.3241,218.148],[347.337,-46.5856,218.152],[346.328,-45.9985,218.158],[345.319,-44.9732,218.159],[344.243,-44.0985,218.151],[343.187,-42.9305,218.149],[342.157,-42.7851,218.144],[341.097,-41.4677,218.145],[340.046,-40.0006,218.147],[339.014,-39.9967,218.153],[337.969,-39.9951,218.152],[336.914,-39.9978,218.148],[335.866,-40,218.144],[334.859,-40.003,218.141],[344.243,-44.0985,218.151],[343.187,-42.9305,218.149],[342.157,-42.7851,218.144],[341.097,-41.4677,218.145],[340.046,-40.0006,218.147],[339.014,-39.9967,218.153],[337.969,-39.9951,218.152],[336.914,-39.9978,218.148],[335.866,-40,218.144],[334.859,-40.003,218.141],[332.054,-39.994,188.152],[0,0,0],[0,0,0],[0,0,0],[0,0,0],[0,0,0],[0,0,0],[0,0,0],[0,0,0],[0,0,0]];
    TASK PERS robtarget robtSSBPeripheryCenter:=[[380.016,59.3683,158.112],[0.707091,0.707123,2.86463E-05,1.00975E-05],[-1,-1,1,1],[4837,9E+09,9E+09,9E+09,9E+09,9E+09]];
    TASK PERS pose poseSSBPeripheryCenter:=[[0.0264893,2.21828,-0.0381012],[1,0,0,0]];

    !Scan saddle header points
    TASK PERS robtarget robtSSHLaserSmarTacs{20}:=[[[296.85,108.15,0],[3.09086E-08,-3.09086E-08,0.707107,-0.707107],[-1,-1,-1,1],[4838,9E+09,9E+09,9E+09,9E+09,9E+09]],[[296.85,107.225,14.1164],[2.88209E-08,-3.2864E-08,0.75184,-0.659346],[-1,-1,-1,1],[4838,9E+09,9E+09,9E+09,9E+09,9E+09]],[[296.85,104.465,27.9913],[2.66098E-08,-3.46786E-08,0.793353,-0.608761],[-1,-1,-1,1],[4838,9E+09,9E+09,9E+09,9E+09,9E+09]],[[296.85,99.9176,41.3872],[2.42847E-08,-3.63447E-08,0.83147,-0.55557],[-1,-1,-1,1],[4838,9E+09,9E+09,9E+09,9E+09,9E+09]],[[296.85,93.6606,54.075],[2.18557E-08,-3.78552E-08,0.866025,-0.5],[-1,-1,-1,1],[4838,9E+09,9E+09,9E+09,9E+09,9E+09]],[[296.85,85.8012,65.8375],[1.93331E-08,-3.92036E-08,0.896873,-0.442289],[-1,-1,-1,1],[4838,9E+09,9E+09,9E+09,9E+09,9E+09]],[[296.85,76.4736,76.4736],[1.67276E-08,-4.03841E-08,0.92388,-0.382683],[-1,-1,-1,1],[4838,9E+09,9E+09,9E+09,9E+09,9E+09]],[[296.85,65.8375,85.8012],[1.40506E-08,-4.13916E-08,0.94693,-0.321439],[-1,-1,-1,1],[4838,9E+09,9E+09,9E+09,9E+09,9E+09]],[[296.85,54.075,93.6607],[1.13133E-08,-4.2222E-08,0.965926,-0.258819],[-1,0,-2,0],[4838,9E+09,9E+09,9E+09,9E+09,9E+09]],[[296.85,41.3872,99.9176],[8.52767E-09,-4.28715E-08,0.980785,-0.19509],[-1,0,-2,0],[4838,9E+09,9E+09,9E+09,9E+09,9E+09]],[[296.85,27.9913,104.465],[5.70548E-09,-4.33374E-08,0.991445,-0.130526],[-1,0,-2,0],[4838,9E+09,9E+09,9E+09,9E+09,9E+09]],[[296.85,14.1164,107.225],[2.85886E-09,-4.36178E-08,0.997859,-0.0654032],[-1,0,-2,0],[4838,9E+09,9E+09,9E+09,9E+09,9E+09]],[[296.85,-4.72739E-06,108.15],[1.91069E-15,4.37114E-08,-1,-4.37114E-08],[-1,0,-2,0],[4838,9E+09,9E+09,9E+09,9E+09,9E+09]],[[652.53,-493.33,1047.99],[0.459259,-0.544323,-0.447932,-0.54051],[-1,0,-2,0],[4837,9E+09,9E+09,9E+09,9E+09,9E+09]],[[652.53,-493.33,1047.99],[0.459259,-0.544323,-0.447932,-0.54051],[-1,0,-2,1],[4837,9E+09,9E+09,9E+09,9E+09,9E+09]],[[652.53,-493.33,1047.99],[0.459259,-0.544323,-0.447932,-0.54051],[-1,0,-2,1],[4837,9E+09,9E+09,9E+09,9E+09,9E+09]],[[652.53,-493.33,1047.99],[0.459259,-0.544323,-0.447932,-0.54051],[-1,0,-2,1],[4837,9E+09,9E+09,9E+09,9E+09,9E+09]],[[652.53,-493.33,1047.99],[0.459259,-0.544323,-0.447932,-0.54051],[-1,0,-2,1],[4837,9E+09,9E+09,9E+09,9E+09,9E+09]],[[652.53,-493.33,1047.99],[0.459259,-0.544323,-0.447932,-0.54051],[-1,0,-2,1],[4837,9E+09,9E+09,9E+09,9E+09,9E+09]],[[652.53,-493.33,1047.99],[0.459259,-0.544323,-0.447932,-0.54051],[-1,0,-2,1],[4837,9E+09,9E+09,9E+09,9E+09,9E+09]]];
    TASK PERS robtarget robtSSHWireSmarTacs{20}:=[[[296.85,108.15,0],[0.5,0.5,-0.5,0.5],[-1,-1,2,1],[4838,9E+09,9E+09,9E+09,9E+09,9E+09]],[[296.85,107.225,14.1164],[0.466228,0.531631,-0.531631,0.466228],[-1,-1,2,1],[4838,9E+09,9E+09,9E+09,9E+09,9E+09]],[[296.85,104.465,27.9913],[0.430459,0.560986,-0.560986,0.430459],[-1,-1,2,1],[4838,9E+09,9E+09,9E+09,9E+09,9E+09]],[[296.85,99.9176,41.3872],[0.392847,0.587938,-0.587938,0.392848],[-1,0,1,0],[4838,9E+09,9E+09,9E+09,9E+09,9E+09]],[[296.85,93.6606,54.075],[0.353553,0.612372,-0.612372,0.353553],[-1,0,1,0],[4838,9E+09,9E+09,9E+09,9E+09,9E+09]],[[296.85,85.8012,65.8375],[0.312745,0.634185,-0.634185,0.312745],[-1,0,1,0],[4838,9E+09,9E+09,9E+09,9E+09,9E+09]],[[296.85,76.4736,76.4736],[0.270598,0.653282,0.653281,-0.270598],[-1,-1,0,1],[4838,9E+09,9E+09,9E+09,9E+09,9E+09]],[[296.85,65.8375,85.8012],[0.227292,0.669581,0.669581,-0.227292],[-1,-1,0,1],[4838,9E+09,9E+09,9E+09,9E+09,9E+09]],[[296.85,54.075,93.6607],[0.183013,0.683013,0.683013,-0.183013],[-1,-1,0,1],[4838,9E+09,9E+09,9E+09,9E+09,9E+09]],[[296.85,41.3872,99.9176],[0.13795,0.69352,0.69352,-0.13795],[-1,-1,0,1],[4838,9E+09,9E+09,9E+09,9E+09,9E+09]],[[296.85,27.9913,104.465],[0.092296,0.701057,0.701057,-0.092296],[-1,-1,0,1],[4838,9E+09,9E+09,9E+09,9E+09,9E+09]],[[296.85,14.1164,107.225],[0.046247,0.705593,0.705593,-0.046247],[-1,0,-1,0],[4838,9E+09,9E+09,9E+09,9E+09,9E+09]],[[296.85,-4.72739E-06,108.15],[3.09086E-08,-0.707107,-0.707107,-3.09086E-08],[-1,0,-1,0],[4838,9E+09,9E+09,9E+09,9E+09,9E+09]],[[652.53,-493.33,1047.99],[0.459259,-0.544323,-0.447932,-0.54051],[-1,0,-1,0],[4837,9E+09,9E+09,9E+09,9E+09,9E+09]],[[652.53,-493.33,1047.99],[0.459259,-0.544323,-0.447932,-0.54051],[-1,0,-2,1],[4837,9E+09,9E+09,9E+09,9E+09,9E+09]],[[652.53,-493.33,1047.99],[0.459259,-0.544323,-0.447932,-0.54051],[-1,0,-2,1],[4837,9E+09,9E+09,9E+09,9E+09,9E+09]],[[652.53,-493.33,1047.99],[0.459259,-0.544323,-0.447932,-0.54051],[-1,0,-2,1],[4837,9E+09,9E+09,9E+09,9E+09,9E+09]],[[652.53,-493.33,1047.99],[0.459259,-0.544323,-0.447932,-0.54051],[-1,0,-2,1],[4837,9E+09,9E+09,9E+09,9E+09,9E+09]],[[652.53,-493.33,1047.99],[0.459259,-0.544323,-0.447932,-0.54051],[-1,0,-2,1],[4837,9E+09,9E+09,9E+09,9E+09,9E+09]],[[652.53,-493.33,1047.99],[0.459259,-0.544323,-0.447932,-0.54051],[-1,0,-2,1],[4837,9E+09,9E+09,9E+09,9E+09,9E+09]]];
    TASK PERS robtarget robtSSHLinerFrom:=[[452.15,78.15,88.5913],[0.5,0.5,-0.5,0.5],[-1,-1,-1,1],[4837,9E+09,9E+09,9E+09,9E+09,9E+09]];
    TASK PERS robtarget robtSSHLinerTo:=[[452.15,78.15,-88.5913],[0.5,0.5,-0.5,0.5],[-1,-1,-1,1],[4837,9E+09,9E+09,9E+09,9E+09,9E+09]];

    !Scan saddle header results, shared for all the four scan methods
    TASK PERS pose poseSSHs{20}:=[[[-0.0262756,-1.74011,-0.0842074],[1,0,0,0]],[[0.00857544,-1.63525,-0.318074],[1,0,0,0]],[[-0.028656,-1.64377,-0.546583],[1,0,0,0]],[[0.0638428,-2.0858,-0.993671],[1,0,0,0]],[[0.0242615,-5.82465,-3.91956],[1,0,0,0]],[[-0.00445557,-2.85303,-2.25892],[1,0,0,0]],[[-0.0636902,-4.71622,-4.46343],[1,0,0,0]],[[-0.0174561,-1.48105,-1.78532],[1,0,0,0]],[[-0.0214844,-1.60992,-2.29945],[1,0,0,0]],[[-0.0274048,-2.24935,-4.57064],[1,0,0,0]],[[0.00231934,-0.64773,-2.24944],[1,0,0,0]],[[-0.0207214,-0.326895,-2.32129],[1,0,0,0]],[[-0.0108948,0.00979681,-3.05504],[1,0,0,0]],[[0,0,0],[1,0,0,0]],[[0,0,0],[1,0,0,0]],[[0,0,0],[1,0,0,0]],[[0,0,0],[1,0,0,0]],[[0,0,0],[1,0,0,0]],[[0,0,0],[1,0,0,0]],[[0,0,0],[1,0,0,0]]];
    TASK PERS num numSSHLaserValues{100}:=[0,0,0,0,0,0,0,0,0,0,0,0,0,0,0,0,0,0,0,0,0,0,0,0,0,0,0,0,0,0,0,0,0,0,0,0,0,0,0,0,0,0,0,0,0,0,0,0,0,0,0,0,0,0,0,0,0,0,0,0,0,0,0,0,0,0,0,0,0,0,0,0,0,0,0,0,0,0,0,0,0,0,0,0,0,0,0,0,0,0,0,0,0,0,0,0,0,0,0,0];
    TASK PERS robtarget robtSSHPeripherys{100}:=[[[296.824,106.41,-0.0842074],[0.499958,0.500028,-0.500074,0.49994],[-1,-1,2,1],[4838,9E+09,9E+09,9E+09,9E+09,9E+09]],[[296.859,105.59,13.7983],[0.466186,0.531648,-0.531681,0.466194],[-1,-1,2,1],[4838,9E+09,9E+09,9E+09,9E+09,9E+09]],[[296.821,102.821,27.4447],[0.430412,0.561012,-0.561049,0.430389],[-1,-1,2,1],[4838,9E+09,9E+09,9E+09,9E+09,9E+09]],[[296.914,97.8318,40.3935],[0.392741,0.587978,-0.587986,0.392822],[-1,0,1,0],[4838,9E+09,9E+09,9E+09,9E+09,9E+09]],[[296.874,87.836,50.1554],[0.353284,0.612457,-0.612578,0.353322],[-1,0,1,0],[4838,9E+09,9E+09,9E+09,9E+09,9E+09]],[[296.846,82.9481,63.5786],[0.312722,0.634193,-0.634199,0.312722],[-1,0,1,0],[4838,9E+09,9E+09,9E+09,9E+09,9E+09]],[[296.786,71.7574,72.0102],[0.270652,0.653251,0.653232,-0.270739],[-1,-1,0,1],[4838,9E+09,9E+09,9E+09,9E+09,9E+09]],[[296.833,64.3565,84.0158],[0.227343,0.669554,0.669563,-0.227371],[-1,-1,0,1],[4838,9E+09,9E+09,9E+09,9E+09,9E+09]],[[296.829,52.4651,91.3612],[0.183138,0.682977,0.682975,-0.183162],[-1,-1,0,1],[4838,9E+09,9E+09,9E+09,9E+09,9E+09]],[[296.823,39.1379,95.3469],[0.138102,0.693464,0.693504,-0.138156],[-1,-1,0,1],[4838,9E+09,9E+09,9E+09,9E+09,9E+09]],[[296.852,27.3436,102.215],[0.092318,0.70103,0.701076,-0.0923436],[-1,-1,0,1],[4838,9E+09,9E+09,9E+09,9E+09,9E+09]],[[296.829,13.7895,104.903],[0.0462517,0.705607,0.705577,-0.0462699],[-1,0,-1,0],[4838,9E+09,9E+09,9E+09,9E+09,9E+09]],[[296.839,0.00979208,105.095],[2.40556E-05,-0.707095,-0.707119,-6.38552E-07],[-1,0,-1,0],[4838,9E+09,9E+09,9E+09,9E+09,9E+09]],[[75.54,-110.49,75.53],[0.104911,-0.592891,0.59209,0.535634],[-1,-2,0,1],[3747.5,9E+09,9E+09,9E+09,9E+09,9E+09]],[[75.54,-110.49,75.53],[0.104911,-0.592891,0.59209,0.535634],[-1,0,-1,0],[3747.5,9E+09,9E+09,9E+09,9E+09,9E+09]],[[75.54,-110.49,75.53],[0.104911,-0.592891,0.59209,0.535634],[-1,0,-1,0],[3747.5,9E+09,9E+09,9E+09,9E+09,9E+09]],[[75.54,-110.49,75.53],[0.104911,-0.592891,0.59209,0.535634],[-1,0,-1,0],[3747.5,9E+09,9E+09,9E+09,9E+09,9E+09]],[[75.54,-110.49,75.53],[0.104911,-0.592891,0.59209,0.535634],[-1,0,-1,0],[3747.5,9E+09,9E+09,9E+09,9E+09,9E+09]],[[75.54,-110.49,75.53],[0.104911,-0.592891,0.59209,0.535634],[-1,0,-1,0],[3747.5,9E+09,9E+09,9E+09,9E+09,9E+09]],[[75.54,-110.49,75.53],[0.104911,-0.592891,0.59209,0.535634],[-1,0,-1,0],[3747.5,9E+09,9E+09,9E+09,9E+09,9E+09]],[[75.54,-110.49,75.53],[0.104911,-0.592891,0.59209,0.535634],[-1,0,-1,0],[3747.5,9E+09,9E+09,9E+09,9E+09,9E+09]],[[75.54,-110.49,75.53],[0.104911,-0.592891,0.59209,0.535634],[-1,0,-1,0],[3747.5,9E+09,9E+09,9E+09,9E+09,9E+09]],[[75.54,-110.49,75.53],[0.104911,-0.592891,0.59209,0.535634],[-1,0,-1,0],[3747.5,9E+09,9E+09,9E+09,9E+09,9E+09]],[[75.54,-110.49,75.53],[0.104911,-0.592891,0.59209,0.535634],[-1,0,-1,0],[3747.5,9E+09,9E+09,9E+09,9E+09,9E+09]],[[75.54,-110.49,75.53],[0.104911,-0.592891,0.59209,0.535634],[-1,0,-1,0],[3747.5,9E+09,9E+09,9E+09,9E+09,9E+09]],[[75.54,-110.49,75.53],[0.104911,-0.592891,0.59209,0.535634],[-1,0,-1,0],[3747.5,9E+09,9E+09,9E+09,9E+09,9E+09]],[[75.54,-110.49,75.53],[0.104911,-0.592891,0.59209,0.535634],[-1,0,-1,0],[3747.5,9E+09,9E+09,9E+09,9E+09,9E+09]],[[75.54,-110.49,75.53],[0.104911,-0.592891,0.59209,0.535634],[-1,0,-1,0],[3747.5,9E+09,9E+09,9E+09,9E+09,9E+09]],[[75.54,-110.49,75.53],[0.104911,-0.592891,0.59209,0.535634],[-1,0,-1,0],[3747.5,9E+09,9E+09,9E+09,9E+09,9E+09]],[[75.54,-110.49,75.53],[0.104911,-0.592891,0.59209,0.535634],[-1,0,-1,0],[3747.5,9E+09,9E+09,9E+09,9E+09,9E+09]],[[75.54,-110.49,75.53],[0.104911,-0.592891,0.59209,0.535634],[-1,0,-1,0],[3747.5,9E+09,9E+09,9E+09,9E+09,9E+09]],[[75.54,-110.49,75.53],[0.104911,-0.592891,0.59209,0.535634],[-1,0,-1,0],[3747.5,9E+09,9E+09,9E+09,9E+09,9E+09]],[[75.54,-110.49,75.53],[0.104911,-0.592891,0.59209,0.535634],[-1,0,-1,0],[3747.5,9E+09,9E+09,9E+09,9E+09,9E+09]],[[75.54,-110.49,75.53],[0.104911,-0.592891,0.59209,0.535634],[-1,0,-1,0],[3747.5,9E+09,9E+09,9E+09,9E+09,9E+09]],[[75.54,-110.49,75.53],[0.104911,-0.592891,0.59209,0.535634],[-1,0,-1,0],[3747.5,9E+09,9E+09,9E+09,9E+09,9E+09]],[[75.54,-110.49,75.53],[0.104911,-0.592891,0.59209,0.535634],[-1,0,-1,0],[3747.5,9E+09,9E+09,9E+09,9E+09,9E+09]],[[75.54,-110.49,75.53],[0.104911,-0.592891,0.59209,0.535634],[-1,0,-1,0],[3747.5,9E+09,9E+09,9E+09,9E+09,9E+09]],[[75.54,-110.49,75.53],[0.104911,-0.592891,0.59209,0.535634],[-1,0,-1,0],[3747.5,9E+09,9E+09,9E+09,9E+09,9E+09]],[[75.54,-110.49,75.53],[0.104911,-0.592891,0.59209,0.535634],[-1,0,-1,0],[3747.5,9E+09,9E+09,9E+09,9E+09,9E+09]],[[75.54,-110.49,75.53],[0.104911,-0.592891,0.59209,0.535634],[-1,0,-1,0],[3747.5,9E+09,9E+09,9E+09,9E+09,9E+09]],[[75.54,-110.49,75.53],[0.104911,-0.592891,0.59209,0.535634],[-1,0,-1,0],[3747.5,9E+09,9E+09,9E+09,9E+09,9E+09]],[[75.54,-110.49,75.53],[0.104911,-0.592891,0.59209,0.535634],[-1,0,-1,0],[3747.5,9E+09,9E+09,9E+09,9E+09,9E+09]],[[75.54,-110.49,75.53],[0.104911,-0.592891,0.59209,0.535634],[-1,0,-1,0],[3747.5,9E+09,9E+09,9E+09,9E+09,9E+09]],[[75.54,-110.49,75.53],[0.104911,-0.592891,0.59209,0.535634],[-1,0,-1,0],[3747.5,9E+09,9E+09,9E+09,9E+09,9E+09]],[[75.54,-110.49,75.53],[0.104911,-0.592891,0.59209,0.535634],[-1,0,-1,0],[3747.5,9E+09,9E+09,9E+09,9E+09,9E+09]],[[75.54,-110.49,75.53],[0.104911,-0.592891,0.59209,0.535634],[-1,0,-1,0],[3747.5,9E+09,9E+09,9E+09,9E+09,9E+09]],[[75.54,-110.49,75.53],[0.104911,-0.592891,0.59209,0.535634],[-1,0,-1,0],[3747.5,9E+09,9E+09,9E+09,9E+09,9E+09]],[[75.54,-110.49,75.53],[0.104911,-0.592891,0.59209,0.535634],[-1,0,-1,0],[3747.5,9E+09,9E+09,9E+09,9E+09,9E+09]],[[75.54,-110.49,75.53],[0.104911,-0.592891,0.59209,0.535634],[-1,0,-1,0],[3747.5,9E+09,9E+09,9E+09,9E+09,9E+09]],[[75.54,-110.49,75.53],[0.104911,-0.592891,0.59209,0.535634],[-1,0,-1,0],[3747.5,9E+09,9E+09,9E+09,9E+09,9E+09]],[[75.54,-110.49,75.53],[0.104911,-0.592891,0.59209,0.535634],[-1,0,-1,0],[3747.5,9E+09,9E+09,9E+09,9E+09,9E+09]],[[75.54,-110.49,75.53],[0.104911,-0.592891,0.59209,0.535634],[-1,0,-1,0],[3747.5,9E+09,9E+09,9E+09,9E+09,9E+09]],[[75.54,-110.49,75.53],[0.104911,-0.592891,0.59209,0.535634],[-1,0,-1,0],[3747.5,9E+09,9E+09,9E+09,9E+09,9E+09]],[[75.54,-110.49,75.53],[0.104911,-0.592891,0.59209,0.535634],[-1,0,-1,0],[3747.5,9E+09,9E+09,9E+09,9E+09,9E+09]],[[75.54,-110.49,75.53],[0.104911,-0.592891,0.59209,0.535634],[-1,0,-1,0],[3747.5,9E+09,9E+09,9E+09,9E+09,9E+09]],[[75.54,-110.49,75.53],[0.104911,-0.592891,0.59209,0.535634],[-1,0,-1,0],[3747.5,9E+09,9E+09,9E+09,9E+09,9E+09]],[[75.54,-110.49,75.53],[0.104911,-0.592891,0.59209,0.535634],[-1,0,-1,0],[3747.5,9E+09,9E+09,9E+09,9E+09,9E+09]],[[75.54,-110.49,75.53],[0.104911,-0.592891,0.59209,0.535634],[-1,0,-1,0],[3747.5,9E+09,9E+09,9E+09,9E+09,9E+09]],[[75.54,-110.49,75.53],[0.104911,-0.592891,0.59209,0.535634],[-1,0,-1,0],[3747.5,9E+09,9E+09,9E+09,9E+09,9E+09]],[[75.54,-110.49,75.53],[0.104911,-0.592891,0.59209,0.535634],[-1,0,-1,0],[3747.5,9E+09,9E+09,9E+09,9E+09,9E+09]],[[75.54,-110.49,75.53],[0.104911,-0.592891,0.59209,0.535634],[-1,0,-1,0],[3747.5,9E+09,9E+09,9E+09,9E+09,9E+09]],[[75.54,-110.49,75.53],[0.104911,-0.592891,0.59209,0.535634],[-1,0,-1,0],[3747.5,9E+09,9E+09,9E+09,9E+09,9E+09]],[[75.54,-110.49,75.53],[0.104911,-0.592891,0.59209,0.535634],[-1,0,-1,0],[3747.5,9E+09,9E+09,9E+09,9E+09,9E+09]],[[75.54,-110.49,75.53],[0.104911,-0.592891,0.59209,0.535634],[-1,0,-1,0],[3747.5,9E+09,9E+09,9E+09,9E+09,9E+09]],[[75.54,-110.49,75.53],[0.104911,-0.592891,0.59209,0.535634],[-1,0,-1,0],[3747.5,9E+09,9E+09,9E+09,9E+09,9E+09]],[[75.54,-110.49,75.53],[0.104911,-0.592891,0.59209,0.535634],[-1,0,-1,0],[3747.5,9E+09,9E+09,9E+09,9E+09,9E+09]],[[75.54,-110.49,75.53],[0.104911,-0.592891,0.59209,0.535634],[-1,0,-1,0],[3747.5,9E+09,9E+09,9E+09,9E+09,9E+09]],[[75.54,-110.49,75.53],[0.104911,-0.592891,0.59209,0.535634],[-1,0,-1,0],[3747.5,9E+09,9E+09,9E+09,9E+09,9E+09]],[[75.54,-110.49,75.53],[0.104911,-0.592891,0.59209,0.535634],[-1,0,-1,0],[3747.5,9E+09,9E+09,9E+09,9E+09,9E+09]],[[75.54,-110.49,75.53],[0.104911,-0.592891,0.59209,0.535634],[-1,0,-1,0],[3747.5,9E+09,9E+09,9E+09,9E+09,9E+09]],[[75.54,-110.49,75.53],[0.104911,-0.592891,0.59209,0.535634],[-1,0,-1,0],[3747.5,9E+09,9E+09,9E+09,9E+09,9E+09]],[[75.54,-110.49,75.53],[0.104911,-0.592891,0.59209,0.535634],[-1,0,-1,0],[3747.5,9E+09,9E+09,9E+09,9E+09,9E+09]],[[75.54,-110.49,75.53],[0.104911,-0.592891,0.59209,0.535634],[-1,0,-1,0],[3747.5,9E+09,9E+09,9E+09,9E+09,9E+09]],[[75.54,-110.49,75.53],[0.104911,-0.592891,0.59209,0.535634],[-1,0,-1,0],[3747.5,9E+09,9E+09,9E+09,9E+09,9E+09]],[[75.54,-110.49,75.53],[0.104911,-0.592891,0.59209,0.535634],[-1,0,-1,0],[3747.5,9E+09,9E+09,9E+09,9E+09,9E+09]],[[75.54,-110.49,75.53],[0.104911,-0.592891,0.59209,0.535634],[-1,0,-1,0],[3747.5,9E+09,9E+09,9E+09,9E+09,9E+09]],[[75.54,-110.49,75.53],[0.104911,-0.592891,0.59209,0.535634],[-1,0,-1,0],[3747.5,9E+09,9E+09,9E+09,9E+09,9E+09]],[[75.54,-110.49,75.53],[0.104911,-0.592891,0.59209,0.535634],[-1,0,-1,0],[3747.5,9E+09,9E+09,9E+09,9E+09,9E+09]],[[75.54,-110.49,75.53],[0.104911,-0.592891,0.59209,0.535634],[-1,0,-1,0],[3747.5,9E+09,9E+09,9E+09,9E+09,9E+09]],[[75.54,-110.49,75.53],[0.104911,-0.592891,0.59209,0.535634],[-1,0,-1,0],[3747.5,9E+09,9E+09,9E+09,9E+09,9E+09]],[[75.54,-110.49,75.53],[0.104911,-0.592891,0.59209,0.535634],[-1,0,-1,0],[3747.5,9E+09,9E+09,9E+09,9E+09,9E+09]],[[75.54,-110.49,75.53],[0.104911,-0.592891,0.59209,0.535634],[-1,0,-1,0],[3747.5,9E+09,9E+09,9E+09,9E+09,9E+09]],[[75.54,-110.49,75.53],[0.104911,-0.592891,0.59209,0.535634],[-1,0,-1,0],[3747.5,9E+09,9E+09,9E+09,9E+09,9E+09]],[[75.54,-110.49,75.53],[0.104911,-0.592891,0.59209,0.535634],[-1,0,-1,0],[3747.5,9E+09,9E+09,9E+09,9E+09,9E+09]],[[75.54,-110.49,75.53],[0.104911,-0.592891,0.59209,0.535634],[-1,0,-1,0],[3747.5,9E+09,9E+09,9E+09,9E+09,9E+09]],[[75.54,-110.49,75.53],[0.104911,-0.592891,0.59209,0.535634],[-1,0,-1,0],[3747.5,9E+09,9E+09,9E+09,9E+09,9E+09]],[[75.54,-110.49,75.53],[0.104911,-0.592891,0.59209,0.535634],[-1,0,-1,0],[3747.5,9E+09,9E+09,9E+09,9E+09,9E+09]],[[75.54,-110.49,75.53],[0.104911,-0.592891,0.59209,0.535634],[-1,0,-1,0],[3747.5,9E+09,9E+09,9E+09,9E+09,9E+09]],[[75.54,-110.49,75.53],[0.104911,-0.592891,0.59209,0.535634],[-1,0,-1,0],[3747.5,9E+09,9E+09,9E+09,9E+09,9E+09]],[[75.54,-110.49,75.53],[0.104911,-0.592891,0.59209,0.535634],[-1,0,-1,0],[3747.5,9E+09,9E+09,9E+09,9E+09,9E+09]],[[75.54,-110.49,75.53],[0.104911,-0.592891,0.59209,0.535634],[-1,0,-1,0],[3747.5,9E+09,9E+09,9E+09,9E+09,9E+09]],[[75.54,-110.49,75.53],[0.104911,-0.592891,0.59209,0.535634],[-1,0,-1,0],[3747.5,9E+09,9E+09,9E+09,9E+09,9E+09]],[[75.54,-110.49,75.53],[0.104911,-0.592891,0.59209,0.535634],[-1,0,-1,0],[3747.5,9E+09,9E+09,9E+09,9E+09,9E+09]],[[75.54,-110.49,75.53],[0.104911,-0.592891,0.59209,0.535634],[-1,0,-1,0],[3747.5,9E+09,9E+09,9E+09,9E+09,9E+09]],[[75.54,-110.49,75.53],[0.104911,-0.592891,0.59209,0.535634],[-1,0,-1,0],[3747.5,9E+09,9E+09,9E+09,9E+09,9E+09]],[[75.54,-110.49,75.53],[0.104911,-0.592891,0.59209,0.535634],[-1,0,-1,0],[3747.5,9E+09,9E+09,9E+09,9E+09,9E+09]],[[75.54,-110.49,75.53],[0.104911,-0.592891,0.59209,0.535634],[-1,0,-1,0],[3747.5,9E+09,9E+09,9E+09,9E+09,9E+09]],[[75.54,-110.49,75.53],[0.104911,-0.592891,0.59209,0.535634],[-1,0,-1,0],[3747.5,9E+09,9E+09,9E+09,9E+09,9E+09]],[[75.54,-110.49,75.53],[0.104911,-0.592891,0.59209,0.535634],[-1,0,-1,0],[3747.5,9E+09,9E+09,9E+09,9E+09,9E+09]],[[75.54,-110.49,75.53],[0.104911,-0.592891,0.59209,0.535634],[-1,0,-1,0],[3747.5,9E+09,9E+09,9E+09,9E+09,9E+09]]];
    TASK PERS pos posSSHPeripherys{100}:=[[1189.24,121.652,101.194],[1189.25,123.699,98.2734],[1189.25,126.196,95.1572],[1189.22,101.15,121.436],[1189.22,104.524,118.442],[1189.22,107.745,115.595],[1189.22,110.667,112.689],[1189.22,113.314,109.771],[1189.22,116.535,106.915],[1189.23,119.168,103.959],[1189.24,121.652,101.194],[1189.25,123.699,98.2734],[1189.25,126.196,95.1572],[1189.26,127.954,92.3937],[1189.26,130.439,89.5647],[1189.27,132.657,86.2744],[1189.27,134.276,83.7452],[1189.28,136.015,80.8203],[1189.29,137.934,77.3217],[1189.31,139.385,75.1255],[1189.29,140.697,72.2896],[1189.26,142.452,69.2123],[1189.25,144.2,66.543],[1189.25,145.234,63.5986],[1189.25,146.268,60.7559],[1189.25,147.864,57.7798],[1189.25,148.747,54.9495],[1189.24,149.926,52.044],[1189.24,150.959,49.109],[1189.24,151.977,46.2625],[1189.24,152.571,43.3276],[1189.25,153.298,40.4997],[1189.25,154.014,37.6014],[1189.25,155.204,34.7927],[1189.25,155.778,31.8007],[1189.25,156.359,28.9936],[1189.24,156.814,26.0656],[1189.24,157.394,23.2566],[1189.24,158.118,20.3438],[1189.24,158.119,17.4939],[1189.24,158.42,14.5148],[1189.25,158.698,11.6499],[1189.25,157.393,8.75073],[1189.25,159.449,5.88725],[1189.25,159.151,2.90934],[1189.25,159.45,-0.0296575],[1189.25,159.008,-2.84319],[1189.24,159.148,-5.7465],[1189.24,158.998,-8.53622],[1189.24,159.146,-11.5047],[1189.24,158.987,-14.4503],[1189.24,158.708,-17.4008],[1189.25,158.263,-20.175],[1189.25,158.123,-23.12],[1189.26,157.531,-25.9004],[1189.25,156.804,-28.8832],[1189.25,156.496,-31.703],[1189.25,155.798,-34.6871],[1189.24,155.195,-37.4615],[1189.24,154.325,-40.4037],[1189.24,153.883,-43.2298],[1189.24,152.997,-46.175],[1189.24,151.691,-49.1231],[1189.25,151.247,-51.9159],[1189.26,150.353,-54.83],[1189.26,148.903,-57.76],[1189.26,147.861,-60.5696],[1189.25,147.004,-63.5168],[1189.25,145.535,-66.5052],[1189.24,144.369,-69.3419],[1189.24,142.754,-72.2589],[1189.24,141.149,-75.0635],[1189.24,139.966,-77.9749],[1189.24,138.366,-80.9294],[1189.25,136.601,-83.7217],[1189.26,134.829,-86.6574],[1189.26,133.086,-89.6122],[1189.25,130.876,-92.4367],[1189.25,128.692,-95.4105],[1189.25,126.783,-98.3034],[1189.24,124.74,-101.135],[1189.25,122.69,-104.085],[1189.25,119.609,-106.886],[1189.25,117.42,-109.832],[1189.25,114.327,-112.648],[1189.25,111.701,-115.579],[1189.26,107.736,-118.481],[1189.25,105.547,-121.46],[1189.25,102.483,-124.296],[1189.25,98.3795,-127.233],[297.852,64.3947,-88.033],[0,0,0],[0,0,0],[0,0,0],[0,0,0],[0,0,0],[0,0,0],[0,0,0],[0,0,0],[0,0,0]];
    TASK PERS robtarget robtSSHPeripheryCenter:=[[1189.27,158.927,-1.83617],[0.500019,0.499991,-0.499968,0.500023],[0,0,-2,1],[4202,9E+09,9E+09,9E+09,9E+09,9E+09]];
    TASK PERS pose poseSSHPeripheryCenter:=[[0.0245361,-0.323227,0.0463184],[1,0,0,0]];

    TASK PERS jointtarget jointSSApproach:=[[10.0959,5.51191,52.6931,21.289,-34.0337,-120.075],[4837,9E+09,9E+09,9E+09,9E+09,9E+09]];
    TASK PERS jointtarget jointSSDepart:=[[10.3175,41.3585,56.6399,9.64823,-88.877,-149.089],[4837,9E+09,9E+09,9E+09,9E+09,9E+09]];

    VAR iodev iodevSSBLog;
    VAR iodev iodevSSHLog;

    TASK PERS num numSSHLLSInterval:=0.103616;
    TASK PERS num numSSHLLSScan:=90;
    TASK PERS pos posSSHLLSClosest:=[1189.25,159.449,5.88725];
    TASK PERS num numSSHLLSClosestLaseValue:=-30.2179;
    TASK PERS num numSSHLLSClosestIndex:=44;
    VAR intnum intSSHLinerLaserScan;

    TASK PERS num numSSBLLSInterval:=0.104032;
    TASK PERS num numSSBLLSScan:=90;
    TASK PERS pos posSSBLLSClosest:=[388.11,-58.601,218.152];
    TASK PERS num numSSBLLSClosestLaseValue:=31.3959;
    TASK PERS num numSSBLLSClosestIndex:=39;
    VAR intnum intSSBLinerLaserScan;


    CONST string strSPBLogFileName:="ScanPlatoonBranch2.csv";
    CONST string strSPHLogFileName:="ScanPlatoonHeader2.csv";

    !For platoon branch SmarTac
    TASK PERS num numSPBPointsTotal:=13;
    !Scan platoon branch range
    TASK PERS num numSPBAngleFrom:=140;
    TASK PERS num numSPBAngleTo:=40;

    !For platoon header SmarTac
    TASK PERS num numSPHPointsTotal:=13;
    !Scan platoon header range
    TASK PERS num numSPHAngleFrom:=0;
    TASK PERS num numSPHAngleTo:=60;

    !Scan platoon branch points
    TASK PERS robtarget robtSPBLaserSmarTacs{20}:=[[[3740.81,24.4902,293.7],[0.640856,0.640856,0.298836,0.298836],[-1,-1,1,1],[1447,9E+09,9E+09,9E+09,9E+09,9E+09]],[[3744.67,28.4616,293.7],[0.660875,0.660875,0.251483,0.251483],[-1,-1,1,1],[1447,9E+09,9E+09,9E+09,9E+09,9E+09]],[[3749.06,31.8321,293.7],[0.677401,0.677401,0.202801,0.202801],[-1,-1,1,1],[1447,9E+09,9E+09,9E+09,9E+09,9E+09]],[[3753.9,34.5303,293.7],[0.690346,0.690346,0.153046,0.153046],[-1,-1,1,1],[1447,9E+09,9E+09,9E+09,9E+09,9E+09]],[[3759.07,36.4994,293.7],[0.699641,0.699641,0.102482,0.102482],[-1,-1,1,1],[1447,9E+09,9E+09,9E+09,9E+09,9E+09]],[[3764.48,37.6977,293.7],[0.705238,0.705238,0.051377,0.051377],[-1,-1,1,1],[1447,9E+09,9E+09,9E+09,9E+09,9E+09]],[[3770,38.1,293.7],[0.707107,0.707107,0,0],[-1,-1,1,1],[1447,9E+09,9E+09,9E+09,9E+09,9E+09]],[[3775.52,37.6977,293.7],[0.0513769,-0.0513769,-0.705238,0.705238],[0,0,3,1],[1447,9E+09,9E+09,9E+09,9E+09,9E+09]],[[3780.93,36.4994,293.7],[0.102482,-0.102482,-0.699641,0.699641],[0,0,3,1],[1447,9E+09,9E+09,9E+09,9E+09,9E+09]],[[3786.1,34.5303,293.7],[0.153046,-0.153046,-0.690346,0.690346],[0,0,2,1],[1447,9E+09,9E+09,9E+09,9E+09,9E+09]],[[3790.94,31.8321,293.7],[0.2028,-0.2028,-0.677401,0.677401],[0,0,2,1],[1447,9E+09,9E+09,9E+09,9E+09,9E+09]],[[3795.33,28.4617,293.7],[0.251483,-0.251483,-0.660875,0.660875],[0,0,2,1],[1447,9E+09,9E+09,9E+09,9E+09,9E+09]],[[3799.19,24.4902,293.7],[0.298836,-0.298836,-0.640856,0.640856],[0,0,2,1],[1447,9E+09,9E+09,9E+09,9E+09,9E+09]],[[652.53,-493.33,1047.99],[0.459259,-0.544323,-0.447932,-0.54051],[0,0,2,1],[4837,9E+09,9E+09,9E+09,9E+09,9E+09]],[[652.53,-493.33,1047.99],[0.459259,-0.544323,-0.447932,-0.54051],[-1,0,-2,1],[4837,9E+09,9E+09,9E+09,9E+09,9E+09]],[[652.53,-493.33,1047.99],[0.459259,-0.544323,-0.447932,-0.54051],[-1,0,-2,1],[4837,9E+09,9E+09,9E+09,9E+09,9E+09]],[[652.53,-493.33,1047.99],[0.459259,-0.544323,-0.447932,-0.54051],[-1,0,-2,1],[4837,9E+09,9E+09,9E+09,9E+09,9E+09]],[[652.53,-493.33,1047.99],[0.459259,-0.544323,-0.447932,-0.54051],[-1,0,-2,1],[4837,9E+09,9E+09,9E+09,9E+09,9E+09]],[[652.53,-493.33,1047.99],[0.459259,-0.544323,-0.447932,-0.54051],[-1,0,-2,1],[4837,9E+09,9E+09,9E+09,9E+09,9E+09]],[[652.53,-493.33,1047.99],[0.459259,-0.544323,-0.447932,-0.54051],[-1,0,-2,1],[4837,9E+09,9E+09,9E+09,9E+09,9E+09]]];
    TASK PERS robtarget robtSPBWireSmarTacs{20}:=[[[428.493,28.575,188.15],[0.683013,0.183013,-0.683013,0.183013],[0,1,-3,1],[4838,9E+09,9E+09,9E+09,9E+09,9E+09]],[[422.779,36.7353,188.15],[0.664463,0.241845,-0.664463,0.241845],[0,1,-3,1],[4838,9E+09,9E+09,9E+09,9E+09,9E+09]],[[415.735,43.7794,188.15],[0.640856,0.298836,-0.640856,0.298836],[0,1,-3,1],[4838,9E+09,9E+09,9E+09,9E+09,9E+09]],[[407.575,49.4934,188.15],[0.612372,0.353553,-0.612372,0.353553],[0,0,-3,1],[4838,9E+09,9E+09,9E+09,9E+09,9E+09]],[[398.546,53.7034,188.15],[0.579228,0.40558,-0.579228,0.40558],[0,0,-3,1],[4838,9E+09,9E+09,9E+09,9E+09,9E+09]],[[388.924,56.2818,188.15],[0.541675,0.454519,-0.541675,0.454519],[0,0,-3,1],[4838,9E+09,9E+09,9E+09,9E+09,9E+09]],[[379,57.15,188.15],[0.5,0.5,-0.5,0.5],[0,0,-3,1],[4838,9E+09,9E+09,9E+09,9E+09,9E+09]],[[369.076,56.2818,188.15],[0.454519,0.541675,-0.454519,0.541675],[-1,-1,-2,1],[4838,9E+09,9E+09,9E+09,9E+09,9E+09]],[[359.454,53.7034,188.15],[0.40558,0.579228,-0.40558,0.579228],[-1,-1,-2,1],[4838,9E+09,9E+09,9E+09,9E+09,9E+09]],[[350.425,49.4934,188.15],[0.353553,0.612372,-0.353553,0.612372],[-1,-1,-2,1],[4838,9E+09,9E+09,9E+09,9E+09,9E+09]],[[342.265,43.7794,188.15],[0.298836,0.640856,-0.298836,0.640856],[-1,-2,-2,1],[4838,9E+09,9E+09,9E+09,9E+09,9E+09]],[[335.221,36.7353,188.15],[0.241845,0.664463,-0.241845,0.664463],[-1,-2,-2,1],[4838,9E+09,9E+09,9E+09,9E+09,9E+09]],[[329.507,28.575,188.15],[0.183013,0.683013,-0.183013,0.683013],[-1,-2,-2,1],[4838,9E+09,9E+09,9E+09,9E+09,9E+09]],[[652.53,-493.33,1047.99],[0.459259,-0.544323,-0.447932,-0.54051],[-1,-1,-2,1],[4837,9E+09,9E+09,9E+09,9E+09,9E+09]],[[652.53,-493.33,1047.99],[0.459259,-0.544323,-0.447932,-0.54051],[-1,0,-2,1],[4837,9E+09,9E+09,9E+09,9E+09,9E+09]],[[652.53,-493.33,1047.99],[0.459259,-0.544323,-0.447932,-0.54051],[-1,0,-2,1],[4837,9E+09,9E+09,9E+09,9E+09,9E+09]],[[652.53,-493.33,1047.99],[0.459259,-0.544323,-0.447932,-0.54051],[-1,0,-2,1],[4837,9E+09,9E+09,9E+09,9E+09,9E+09]],[[652.53,-493.33,1047.99],[0.459259,-0.544323,-0.447932,-0.54051],[-1,0,-2,1],[4837,9E+09,9E+09,9E+09,9E+09,9E+09]],[[652.53,-493.33,1047.99],[0.459259,-0.544323,-0.447932,-0.54051],[-1,0,-2,1],[4837,9E+09,9E+09,9E+09,9E+09,9E+09]],[[652.53,-493.33,1047.99],[0.459259,-0.544323,-0.447932,-0.54051],[-1,0,-2,1],[4837,9E+09,9E+09,9E+09,9E+09,9E+09]]];
    TASK PERS robtarget robtSPBLinerFrom:=[[3274.49,38.1,268.15],[0.707107,0.707107,0,0],[0,0,1,1],[1967,9E+09,9E+09,9E+09,9E+09,9E+09]];
    TASK PERS robtarget robtSPBLinerTo:=[[3225.51,38.1,268.15],[0.707107,0.707107,0,0],[0,0,1,1],[1967,9E+09,9E+09,9E+09,9E+09,9E+09]];

    !Scan platoon branch results, shared for all the four scan methods
    TASK PERS pose poseSPBs{20}:=[[[-0.046875,0.0590725,-0.0253296],[1,0,0,0]],[[-0.557373,0.657007,0.0239868],[1,0,0,0]],[[-0.405762,0.598202,-0.00518799],[1,0,0,0]],[[-0.0944824,0.206917,-0.00604248],[1,0,0,0]],[[-0.506836,1.71361,0.0100403],[1,0,0,0]],[[-0.416016,2.88994,0.0373535],[1,0,0,0]],[[0.00732422,1.00344,0.035614],[1,0,0,0]],[[0.331543,2.17712,-0.0392761],[1,0,0,0]],[[0.362305,1.30855,-0.0111084],[1,0,0,0]],[[0.821045,1.83185,0.0217896],[1,0,0,0]],[[1.50269,2.27361,-0.0183105],[1,0,0,0]],[[1.2002,1.41495,-0.0211182],[1,0,0,0]],[[1.10938,0.907724,0.00576782],[1,0,0,0]],[[0,0,0],[1,0,0,0]],[[0,0,0],[1,0,0,0]],[[0,0,0],[1,0,0,0]],[[0,0,0],[1,0,0,0]],[[0,0,0],[1,0,0,0]],[[0,0,0],[1,0,0,0]],[[0,0,0],[1,0,0,0]]];
    TASK PERS num numSPBLaserValues{100}:=[0.038147,0.038147,-0.108337,-0.108337,5.01877,30.517,28.7591,15.4286,-1.28025,1.06357,3.55388,6.92313,9.70641,0,0,0,0,0,0,0,0,0,0,0,0,0,0,0,0,0,0,0,0,0,0,0,0,0,0,0,0,0,0,0,0,0,0,0,0,0,0,0,0,0,0,0,0,0,0,0,0,0,0,0,0,0,0,0,0,0,0,0,0,0,0,0,0,0,0,0,0,0,0,0,0,0,0,0,0,0,0,0,0,0,0,0,0,0,0,0];
    TASK PERS robtarget robtSPBPeripherys{100}:=[[[2245.8,24.5248,268.125],[0.640852,0.640855,0.298848,0.298837],[-1,-1,1,1],[2942,9E+09,9E+09,9E+09,9E+09,9E+09]],[[2249.14,29.0902,268.174],[0.660884,0.660859,0.2515,0.251486],[-1,-1,1,1],[2942,9E+09,9E+09,9E+09,9E+09,9E+09]],[[2253.6,32.5208,268.145],[0.677393,0.677411,0.20279,0.202803],[-1,-1,1,1],[2942,9E+09,9E+09,9E+09,9E+09,9E+09]],[[2258.76,34.8354,268.144],[0.690355,0.690338,0.153046,0.15304],[-1,-1,1,1],[2942,9E+09,9E+09,9E+09,9E+09,9E+09]],[[2265.01,33.4051,268.16],[0.699648,0.699632,0.102491,0.102482],[-1,-1,1,1],[2942,9E+09,9E+09,9E+09,9E+09,9E+09]],[[2273.49,10.393,268.189],[0.705261,0.705214,0.0514384,0.0513308],[-1,-1,1,1],[2942,9E+09,9E+09,9E+09,9E+09,9E+09]],[[2275.01,10.3443,268.188],[0.70713,0.707083,7.83675E-06,3.01479E-06],[-1,-1,1,1],[2942,9E+09,9E+09,9E+09,9E+09,9E+09]],[[2278.62,24.6091,268.11],[0.0513852,-0.051369,-0.705259,0.705216],[0,0,3,1],[2942,9E+09,9E+09,9E+09,9E+09,9E+09]],[[2286.66,39.0344,268.139],[0.102484,-0.102497,-0.699654,0.699625],[0,0,3,1],[2942.01,9E+09,9E+09,9E+09,9E+09,9E+09]],[[2291.47,35.3983,268.172],[0.153062,-0.153067,-0.690326,0.690357],[0,0,2,1],[2942,9E+09,9E+09,9E+09,9E+09,9E+09]],[[2295.49,31.1364,268.131],[0.202778,-0.202809,-0.677423,0.677383],[0,0,2,1],[2942,9E+09,9E+09,9E+09,9E+09,9E+09]],[[2296.93,24.705,268.129],[0.251521,-0.251467,-0.660878,0.660865],[0,0,2,1],[2942,9E+09,9E+09,9E+09,9E+09,9E+09]],[[2297.86,19.1585,268.156],[0.298829,-0.298823,-0.640869,0.640853],[0,0,2,1],[2942,9E+09,9E+09,9E+09,9E+09,9E+09]],[[75.54,-110.49,75.53],[0.104911,-0.592891,0.59209,0.535634],[-1,-2,0,1],[3747.5,9E+09,9E+09,9E+09,9E+09,9E+09]],[[75.54,-110.49,75.53],[0.104911,-0.592891,0.59209,0.535634],[-1,0,-1,0],[3747.5,9E+09,9E+09,9E+09,9E+09,9E+09]],[[75.54,-110.49,75.53],[0.104911,-0.592891,0.59209,0.535634],[-1,0,-1,0],[3747.5,9E+09,9E+09,9E+09,9E+09,9E+09]],[[75.54,-110.49,75.53],[0.104911,-0.592891,0.59209,0.535634],[-1,0,-1,0],[3747.5,9E+09,9E+09,9E+09,9E+09,9E+09]],[[75.54,-110.49,75.53],[0.104911,-0.592891,0.59209,0.535634],[-1,0,-1,0],[3747.5,9E+09,9E+09,9E+09,9E+09,9E+09]],[[75.54,-110.49,75.53],[0.104911,-0.592891,0.59209,0.535634],[-1,0,-1,0],[3747.5,9E+09,9E+09,9E+09,9E+09,9E+09]],[[75.54,-110.49,75.53],[0.104911,-0.592891,0.59209,0.535634],[-1,0,-1,0],[3747.5,9E+09,9E+09,9E+09,9E+09,9E+09]],[[75.54,-110.49,75.53],[0.104911,-0.592891,0.59209,0.535634],[-1,0,-1,0],[3747.5,9E+09,9E+09,9E+09,9E+09,9E+09]],[[75.54,-110.49,75.53],[0.104911,-0.592891,0.59209,0.535634],[-1,0,-1,0],[3747.5,9E+09,9E+09,9E+09,9E+09,9E+09]],[[75.54,-110.49,75.53],[0.104911,-0.592891,0.59209,0.535634],[-1,0,-1,0],[3747.5,9E+09,9E+09,9E+09,9E+09,9E+09]],[[75.54,-110.49,75.53],[0.104911,-0.592891,0.59209,0.535634],[-1,0,-1,0],[3747.5,9E+09,9E+09,9E+09,9E+09,9E+09]],[[75.54,-110.49,75.53],[0.104911,-0.592891,0.59209,0.535634],[-1,0,-1,0],[3747.5,9E+09,9E+09,9E+09,9E+09,9E+09]],[[75.54,-110.49,75.53],[0.104911,-0.592891,0.59209,0.535634],[-1,0,-1,0],[3747.5,9E+09,9E+09,9E+09,9E+09,9E+09]],[[75.54,-110.49,75.53],[0.104911,-0.592891,0.59209,0.535634],[-1,0,-1,0],[3747.5,9E+09,9E+09,9E+09,9E+09,9E+09]],[[75.54,-110.49,75.53],[0.104911,-0.592891,0.59209,0.535634],[-1,0,-1,0],[3747.5,9E+09,9E+09,9E+09,9E+09,9E+09]],[[75.54,-110.49,75.53],[0.104911,-0.592891,0.59209,0.535634],[-1,0,-1,0],[3747.5,9E+09,9E+09,9E+09,9E+09,9E+09]],[[75.54,-110.49,75.53],[0.104911,-0.592891,0.59209,0.535634],[-1,0,-1,0],[3747.5,9E+09,9E+09,9E+09,9E+09,9E+09]],[[75.54,-110.49,75.53],[0.104911,-0.592891,0.59209,0.535634],[-1,0,-1,0],[3747.5,9E+09,9E+09,9E+09,9E+09,9E+09]],[[75.54,-110.49,75.53],[0.104911,-0.592891,0.59209,0.535634],[-1,0,-1,0],[3747.5,9E+09,9E+09,9E+09,9E+09,9E+09]],[[75.54,-110.49,75.53],[0.104911,-0.592891,0.59209,0.535634],[-1,0,-1,0],[3747.5,9E+09,9E+09,9E+09,9E+09,9E+09]],[[75.54,-110.49,75.53],[0.104911,-0.592891,0.59209,0.535634],[-1,0,-1,0],[3747.5,9E+09,9E+09,9E+09,9E+09,9E+09]],[[75.54,-110.49,75.53],[0.104911,-0.592891,0.59209,0.535634],[-1,0,-1,0],[3747.5,9E+09,9E+09,9E+09,9E+09,9E+09]],[[75.54,-110.49,75.53],[0.104911,-0.592891,0.59209,0.535634],[-1,0,-1,0],[3747.5,9E+09,9E+09,9E+09,9E+09,9E+09]],[[75.54,-110.49,75.53],[0.104911,-0.592891,0.59209,0.535634],[-1,0,-1,0],[3747.5,9E+09,9E+09,9E+09,9E+09,9E+09]],[[75.54,-110.49,75.53],[0.104911,-0.592891,0.59209,0.535634],[-1,0,-1,0],[3747.5,9E+09,9E+09,9E+09,9E+09,9E+09]],[[75.54,-110.49,75.53],[0.104911,-0.592891,0.59209,0.535634],[-1,0,-1,0],[3747.5,9E+09,9E+09,9E+09,9E+09,9E+09]],[[75.54,-110.49,75.53],[0.104911,-0.592891,0.59209,0.535634],[-1,0,-1,0],[3747.5,9E+09,9E+09,9E+09,9E+09,9E+09]],[[75.54,-110.49,75.53],[0.104911,-0.592891,0.59209,0.535634],[-1,0,-1,0],[3747.5,9E+09,9E+09,9E+09,9E+09,9E+09]],[[75.54,-110.49,75.53],[0.104911,-0.592891,0.59209,0.535634],[-1,0,-1,0],[3747.5,9E+09,9E+09,9E+09,9E+09,9E+09]],[[75.54,-110.49,75.53],[0.104911,-0.592891,0.59209,0.535634],[-1,0,-1,0],[3747.5,9E+09,9E+09,9E+09,9E+09,9E+09]],[[75.54,-110.49,75.53],[0.104911,-0.592891,0.59209,0.535634],[-1,0,-1,0],[3747.5,9E+09,9E+09,9E+09,9E+09,9E+09]],[[75.54,-110.49,75.53],[0.104911,-0.592891,0.59209,0.535634],[-1,0,-1,0],[3747.5,9E+09,9E+09,9E+09,9E+09,9E+09]],[[75.54,-110.49,75.53],[0.104911,-0.592891,0.59209,0.535634],[-1,0,-1,0],[3747.5,9E+09,9E+09,9E+09,9E+09,9E+09]],[[75.54,-110.49,75.53],[0.104911,-0.592891,0.59209,0.535634],[-1,0,-1,0],[3747.5,9E+09,9E+09,9E+09,9E+09,9E+09]],[[75.54,-110.49,75.53],[0.104911,-0.592891,0.59209,0.535634],[-1,0,-1,0],[3747.5,9E+09,9E+09,9E+09,9E+09,9E+09]],[[75.54,-110.49,75.53],[0.104911,-0.592891,0.59209,0.535634],[-1,0,-1,0],[3747.5,9E+09,9E+09,9E+09,9E+09,9E+09]],[[75.54,-110.49,75.53],[0.104911,-0.592891,0.59209,0.535634],[-1,0,-1,0],[3747.5,9E+09,9E+09,9E+09,9E+09,9E+09]],[[75.54,-110.49,75.53],[0.104911,-0.592891,0.59209,0.535634],[-1,0,-1,0],[3747.5,9E+09,9E+09,9E+09,9E+09,9E+09]],[[75.54,-110.49,75.53],[0.104911,-0.592891,0.59209,0.535634],[-1,0,-1,0],[3747.5,9E+09,9E+09,9E+09,9E+09,9E+09]],[[75.54,-110.49,75.53],[0.104911,-0.592891,0.59209,0.535634],[-1,0,-1,0],[3747.5,9E+09,9E+09,9E+09,9E+09,9E+09]],[[75.54,-110.49,75.53],[0.104911,-0.592891,0.59209,0.535634],[-1,0,-1,0],[3747.5,9E+09,9E+09,9E+09,9E+09,9E+09]],[[75.54,-110.49,75.53],[0.104911,-0.592891,0.59209,0.535634],[-1,0,-1,0],[3747.5,9E+09,9E+09,9E+09,9E+09,9E+09]],[[75.54,-110.49,75.53],[0.104911,-0.592891,0.59209,0.535634],[-1,0,-1,0],[3747.5,9E+09,9E+09,9E+09,9E+09,9E+09]],[[75.54,-110.49,75.53],[0.104911,-0.592891,0.59209,0.535634],[-1,0,-1,0],[3747.5,9E+09,9E+09,9E+09,9E+09,9E+09]],[[75.54,-110.49,75.53],[0.104911,-0.592891,0.59209,0.535634],[-1,0,-1,0],[3747.5,9E+09,9E+09,9E+09,9E+09,9E+09]],[[75.54,-110.49,75.53],[0.104911,-0.592891,0.59209,0.535634],[-1,0,-1,0],[3747.5,9E+09,9E+09,9E+09,9E+09,9E+09]],[[75.54,-110.49,75.53],[0.104911,-0.592891,0.59209,0.535634],[-1,0,-1,0],[3747.5,9E+09,9E+09,9E+09,9E+09,9E+09]],[[75.54,-110.49,75.53],[0.104911,-0.592891,0.59209,0.535634],[-1,0,-1,0],[3747.5,9E+09,9E+09,9E+09,9E+09,9E+09]],[[75.54,-110.49,75.53],[0.104911,-0.592891,0.59209,0.535634],[-1,0,-1,0],[3747.5,9E+09,9E+09,9E+09,9E+09,9E+09]],[[75.54,-110.49,75.53],[0.104911,-0.592891,0.59209,0.535634],[-1,0,-1,0],[3747.5,9E+09,9E+09,9E+09,9E+09,9E+09]],[[75.54,-110.49,75.53],[0.104911,-0.592891,0.59209,0.535634],[-1,0,-1,0],[3747.5,9E+09,9E+09,9E+09,9E+09,9E+09]],[[75.54,-110.49,75.53],[0.104911,-0.592891,0.59209,0.535634],[-1,0,-1,0],[3747.5,9E+09,9E+09,9E+09,9E+09,9E+09]],[[75.54,-110.49,75.53],[0.104911,-0.592891,0.59209,0.535634],[-1,0,-1,0],[3747.5,9E+09,9E+09,9E+09,9E+09,9E+09]],[[75.54,-110.49,75.53],[0.104911,-0.592891,0.59209,0.535634],[-1,0,-1,0],[3747.5,9E+09,9E+09,9E+09,9E+09,9E+09]],[[75.54,-110.49,75.53],[0.104911,-0.592891,0.59209,0.535634],[-1,0,-1,0],[3747.5,9E+09,9E+09,9E+09,9E+09,9E+09]],[[75.54,-110.49,75.53],[0.104911,-0.592891,0.59209,0.535634],[-1,0,-1,0],[3747.5,9E+09,9E+09,9E+09,9E+09,9E+09]],[[75.54,-110.49,75.53],[0.104911,-0.592891,0.59209,0.535634],[-1,0,-1,0],[3747.5,9E+09,9E+09,9E+09,9E+09,9E+09]],[[75.54,-110.49,75.53],[0.104911,-0.592891,0.59209,0.535634],[-1,0,-1,0],[3747.5,9E+09,9E+09,9E+09,9E+09,9E+09]],[[75.54,-110.49,75.53],[0.104911,-0.592891,0.59209,0.535634],[-1,0,-1,0],[3747.5,9E+09,9E+09,9E+09,9E+09,9E+09]],[[75.54,-110.49,75.53],[0.104911,-0.592891,0.59209,0.535634],[-1,0,-1,0],[3747.5,9E+09,9E+09,9E+09,9E+09,9E+09]],[[75.54,-110.49,75.53],[0.104911,-0.592891,0.59209,0.535634],[-1,0,-1,0],[3747.5,9E+09,9E+09,9E+09,9E+09,9E+09]],[[75.54,-110.49,75.53],[0.104911,-0.592891,0.59209,0.535634],[-1,0,-1,0],[3747.5,9E+09,9E+09,9E+09,9E+09,9E+09]],[[75.54,-110.49,75.53],[0.104911,-0.592891,0.59209,0.535634],[-1,0,-1,0],[3747.5,9E+09,9E+09,9E+09,9E+09,9E+09]],[[75.54,-110.49,75.53],[0.104911,-0.592891,0.59209,0.535634],[-1,0,-1,0],[3747.5,9E+09,9E+09,9E+09,9E+09,9E+09]],[[75.54,-110.49,75.53],[0.104911,-0.592891,0.59209,0.535634],[-1,0,-1,0],[3747.5,9E+09,9E+09,9E+09,9E+09,9E+09]],[[75.54,-110.49,75.53],[0.104911,-0.592891,0.59209,0.535634],[-1,0,-1,0],[3747.5,9E+09,9E+09,9E+09,9E+09,9E+09]],[[75.54,-110.49,75.53],[0.104911,-0.592891,0.59209,0.535634],[-1,0,-1,0],[3747.5,9E+09,9E+09,9E+09,9E+09,9E+09]],[[75.54,-110.49,75.53],[0.104911,-0.592891,0.59209,0.535634],[-1,0,-1,0],[3747.5,9E+09,9E+09,9E+09,9E+09,9E+09]],[[75.54,-110.49,75.53],[0.104911,-0.592891,0.59209,0.535634],[-1,0,-1,0],[3747.5,9E+09,9E+09,9E+09,9E+09,9E+09]],[[75.54,-110.49,75.53],[0.104911,-0.592891,0.59209,0.535634],[-1,0,-1,0],[3747.5,9E+09,9E+09,9E+09,9E+09,9E+09]],[[75.54,-110.49,75.53],[0.104911,-0.592891,0.59209,0.535634],[-1,0,-1,0],[3747.5,9E+09,9E+09,9E+09,9E+09,9E+09]],[[75.54,-110.49,75.53],[0.104911,-0.592891,0.59209,0.535634],[-1,0,-1,0],[3747.5,9E+09,9E+09,9E+09,9E+09,9E+09]],[[75.54,-110.49,75.53],[0.104911,-0.592891,0.59209,0.535634],[-1,0,-1,0],[3747.5,9E+09,9E+09,9E+09,9E+09,9E+09]],[[75.54,-110.49,75.53],[0.104911,-0.592891,0.59209,0.535634],[-1,0,-1,0],[3747.5,9E+09,9E+09,9E+09,9E+09,9E+09]],[[75.54,-110.49,75.53],[0.104911,-0.592891,0.59209,0.535634],[-1,0,-1,0],[3747.5,9E+09,9E+09,9E+09,9E+09,9E+09]],[[75.54,-110.49,75.53],[0.104911,-0.592891,0.59209,0.535634],[-1,0,-1,0],[3747.5,9E+09,9E+09,9E+09,9E+09,9E+09]],[[75.54,-110.49,75.53],[0.104911,-0.592891,0.59209,0.535634],[-1,0,-1,0],[3747.5,9E+09,9E+09,9E+09,9E+09,9E+09]],[[75.54,-110.49,75.53],[0.104911,-0.592891,0.59209,0.535634],[-1,0,-1,0],[3747.5,9E+09,9E+09,9E+09,9E+09,9E+09]],[[75.54,-110.49,75.53],[0.104911,-0.592891,0.59209,0.535634],[-1,0,-1,0],[3747.5,9E+09,9E+09,9E+09,9E+09,9E+09]],[[75.54,-110.49,75.53],[0.104911,-0.592891,0.59209,0.535634],[-1,0,-1,0],[3747.5,9E+09,9E+09,9E+09,9E+09,9E+09]],[[75.54,-110.49,75.53],[0.104911,-0.592891,0.59209,0.535634],[-1,0,-1,0],[3747.5,9E+09,9E+09,9E+09,9E+09,9E+09]],[[75.54,-110.49,75.53],[0.104911,-0.592891,0.59209,0.535634],[-1,0,-1,0],[3747.5,9E+09,9E+09,9E+09,9E+09,9E+09]],[[75.54,-110.49,75.53],[0.104911,-0.592891,0.59209,0.535634],[-1,0,-1,0],[3747.5,9E+09,9E+09,9E+09,9E+09,9E+09]],[[75.54,-110.49,75.53],[0.104911,-0.592891,0.59209,0.535634],[-1,0,-1,0],[3747.5,9E+09,9E+09,9E+09,9E+09,9E+09]],[[75.54,-110.49,75.53],[0.104911,-0.592891,0.59209,0.535634],[-1,0,-1,0],[3747.5,9E+09,9E+09,9E+09,9E+09,9E+09]],[[75.54,-110.49,75.53],[0.104911,-0.592891,0.59209,0.535634],[-1,0,-1,0],[3747.5,9E+09,9E+09,9E+09,9E+09,9E+09]],[[75.54,-110.49,75.53],[0.104911,-0.592891,0.59209,0.535634],[-1,0,-1,0],[3747.5,9E+09,9E+09,9E+09,9E+09,9E+09]]];
    TASK PERS pos posSPBPeripherys{100}:=[[3268.45,34.3313,268.078],[3267.8,34.625,268.071],[3267.24,35.0651,268.067],[3266.65,35.0655,268.066],[3266.01,35.3553,268.077],[3265.44,35.2076,268.085],[3264.85,36.0846,268.097],[3264.2,36.2281,268.108],[3263.63,36.52,268.117],[3263.04,36.5203,268.127],[3262.38,36.8109,268.14],[3261.83,36.957,268.146],[3261.24,36.9574,268.148],[3260.58,37.1038,268.147],[3260.02,37.5438,268.149],[3259.42,37.3968,268.149],[3258.78,37.5405,268.151],[3258.21,37.6857,268.153],[3257.6,37.8341,268.152],[3256.96,37.8338,268.151],[3256.39,37.9827,268.149],[3255.8,37.8356,268.15],[3255.18,37.9805,268.152],[3254.6,37.9838,268.148],[3254.01,37.8363,268.15],[3253.36,37.3957,268.151],[3252.79,37.5444,268.151],[3252.18,36.6663,268.152],[3251.43,37.5461,268.151],[3250.97,38.8752,268.151],[3250.36,38.2911,268.151],[3249.73,38.88,268.151],[3249.16,37.5542,268.152],[3248.56,37.8524,268.147],[3247.93,38.7425,268.146],[3247.35,38.0046,268.148],[3246.74,37.7153,268.145],[3246.12,37.7174,268.146],[3245.55,37.5698,268.15],[3244.91,37.5689,268.154],[3244.3,37.4214,268.159],[3243.72,37.1255,268.166],[3243.12,36.9726,268.176],[3242.5,36.9672,268.185],[3241.93,36.8173,268.193],[3241.31,36.6646,268.2],[3240.67,36.5122,268.209],[3240.11,36.5087,268.216],[3239.5,36.5037,268.227],[3238.87,35.6214,268.233],[3238.29,35.0335,268.239],[3237.68,35.6242,268.237],[3237.05,34.8946,268.232],[3236.48,35.0425,268.228],[3235.89,34.8999,268.213],[3235.27,34.3142,268.207],[3234.7,34.1679,268.202],[3234.09,33.4357,268.196],[3233.48,33.2875,268.193],[3232.89,33.1415,268.185],[3232.26,32.4119,268.178],[3231.65,31.8305,268.172],[3231.09,31.537,268.171],[3230.46,31.0946,268.174],[3229.85,31.3879,268.17],[3229.27,30.9498,268.168],[3228.65,29.336,268.168],[3228.06,29.044,268.168],[3227.49,29.0433,268.168],[3226.87,28.3125,268.166],[3226.27,-111.906,268.166],[3225.7,-111.906,268.165],[3231.09,31.537,268.171],[3230.46,31.0946,268.174],[3229.85,31.3879,268.17],[3229.27,30.9498,268.168],[3228.65,29.336,268.168],[3228.06,29.044,268.168],[3227.49,29.0433,268.168],[3226.87,28.3125,268.166],[3226.27,-111.906,268.166],[3225.7,-111.906,268.165],[3272.56,36.9552,268.162],[3271.96,36.9557,268.16],[3271.34,36.8072,268.161],[3270.67,36.6603,268.164],[3270.14,36.5146,268.162],[3269.5,36.0768,268.157],[3268.92,35.6409,268.15],[3268.31,35.6382,268.154],[332.054,-39.994,188.152],[0,0,0],[0,0,0],[0,0,0],[0,0,0],[0,0,0],[0,0,0],[0,0,0],[0,0,0],[0,0,0]];
    TASK PERS robtarget robtSPBPeripheryCenter:=[[3251.93,36.615,268.099],[0.707081,0.707132,2.79942E-06,4.40377E-06],[-1,-1,1,1],[1967,9E+09,9E+09,9E+09,9E+09,9E+09]];
    TASK PERS pose poseSPBPeripheryCenter:=[[0.0100098,-1.48501,-0.051178],[1,0,0,0]];

    !Scan platoon header points
    TASK PERS robtarget robtSPHLaserSmarTacs{20}:=[[[2703.1,133.7,0],[0.5,0.5,0.5,-0.5],[0,0,0,1],[2602,9E+09,9E+09,9E+09,9E+09,9E+09]],[[2703.1,133.191,11.6527],[0.477714,0.521334,0.521334,-0.477714],[0,0,0,1],[2602,9E+09,9E+09,9E+09,9E+09,9E+09]],[[2703.1,131.669,23.2168],[0.454519,0.541675,0.541675,-0.454519],[0,0,0,1],[2602,9E+09,9E+09,9E+09,9E+09,9E+09]],[[2703.1,129.144,34.6041],[0.430459,0.560986,0.560986,-0.430459],[0,0,0,1],[2602,9E+09,9E+09,9E+09,9E+09,9E+09]],[[2703.1,125.637,45.7281],[0.40558,0.579228,0.579228,-0.40558],[0,0,0,1],[2602,9E+09,9E+09,9E+09,9E+09,9E+09]],[[2703.1,121.173,56.5041],[0.379928,0.596368,0.596368,-0.379928],[0,0,0,1],[2602,9E+09,9E+09,9E+09,9E+09,9E+09]],[[2703.1,115.788,66.85],[0.353553,0.612372,0.612372,-0.353553],[0,0,-1,1],[2602,9E+09,9E+09,9E+09,9E+09,9E+09]],[[2703.1,109.521,76.6872],[0.326506,0.627211,0.627211,-0.326506],[0,0,-1,1],[2602,9E+09,9E+09,9E+09,9E+09,9E+09]],[[2703.1,102.42,85.9407],[0.298836,0.640856,0.640856,-0.298836],[0,0,-1,1],[2602,9E+09,9E+09,9E+09,9E+09,9E+09]],[[2703.1,94.5402,94.5402],[0.270598,0.653282,0.653281,-0.270598],[0,0,-1,1],[2602,9E+09,9E+09,9E+09,9E+09,9E+09]],[[2703.1,85.9407,102.42],[0.241845,0.664463,0.664463,-0.241845],[0,0,-1,1],[2602,9E+09,9E+09,9E+09,9E+09,9E+09]],[[2703.1,76.6872,109.521],[0.212631,0.67438,0.67438,-0.212631],[0,1,-2,1],[2602,9E+09,9E+09,9E+09,9E+09,9E+09]],[[2703.1,66.85,115.788],[0.183013,0.683013,0.683013,-0.183013],[0,1,-2,1],[2602,9E+09,9E+09,9E+09,9E+09,9E+09]],[[652.53,-493.33,1047.99],[0.459259,-0.544323,-0.447932,-0.54051],[0,1,-2,1],[4837,9E+09,9E+09,9E+09,9E+09,9E+09]],[[652.53,-493.33,1047.99],[0.459259,-0.544323,-0.447932,-0.54051],[-1,0,-2,1],[4837,9E+09,9E+09,9E+09,9E+09,9E+09]],[[652.53,-493.33,1047.99],[0.459259,-0.544323,-0.447932,-0.54051],[-1,0,-2,1],[4837,9E+09,9E+09,9E+09,9E+09,9E+09]],[[652.53,-493.33,1047.99],[0.459259,-0.544323,-0.447932,-0.54051],[-1,0,-2,1],[4837,9E+09,9E+09,9E+09,9E+09,9E+09]],[[652.53,-493.33,1047.99],[0.459259,-0.544323,-0.447932,-0.54051],[-1,0,-2,1],[4837,9E+09,9E+09,9E+09,9E+09,9E+09]],[[652.53,-493.33,1047.99],[0.459259,-0.544323,-0.447932,-0.54051],[-1,0,-2,1],[4837,9E+09,9E+09,9E+09,9E+09,9E+09]],[[652.53,-493.33,1047.99],[0.459259,-0.544323,-0.447932,-0.54051],[-1,0,-2,1],[4837,9E+09,9E+09,9E+09,9E+09,9E+09]]];
    TASK PERS robtarget robtSPHWireSmarTacs{20}:=[[[296.85,108.15,0],[0.5,0.5,-0.5,0.5],[-1,-1,2,1],[4838,9E+09,9E+09,9E+09,9E+09,9E+09]],[[296.85,107.225,14.1164],[0.466228,0.531631,-0.531631,0.466228],[-1,-1,2,1],[4838,9E+09,9E+09,9E+09,9E+09,9E+09]],[[296.85,104.465,27.9913],[0.430459,0.560986,-0.560986,0.430459],[-1,-1,2,1],[4838,9E+09,9E+09,9E+09,9E+09,9E+09]],[[296.85,99.9176,41.3872],[0.392847,0.587938,-0.587938,0.392848],[-1,0,1,0],[4838,9E+09,9E+09,9E+09,9E+09,9E+09]],[[296.85,93.6606,54.075],[0.353553,0.612372,-0.612372,0.353553],[-1,0,1,0],[4838,9E+09,9E+09,9E+09,9E+09,9E+09]],[[296.85,85.8012,65.8375],[0.312745,0.634185,-0.634185,0.312745],[-1,0,1,0],[4838,9E+09,9E+09,9E+09,9E+09,9E+09]],[[296.85,76.4736,76.4736],[0.270598,0.653282,0.653281,-0.270598],[-1,-1,0,1],[4838,9E+09,9E+09,9E+09,9E+09,9E+09]],[[296.85,65.8375,85.8012],[0.227292,0.669581,0.669581,-0.227292],[-1,-1,0,1],[4838,9E+09,9E+09,9E+09,9E+09,9E+09]],[[296.85,54.075,93.6607],[0.183013,0.683013,0.683013,-0.183013],[-1,-1,0,1],[4838,9E+09,9E+09,9E+09,9E+09,9E+09]],[[296.85,41.3872,99.9176],[0.13795,0.69352,0.69352,-0.13795],[-1,-1,0,1],[4838,9E+09,9E+09,9E+09,9E+09,9E+09]],[[296.85,27.9913,104.465],[0.092296,0.701057,0.701057,-0.092296],[-1,-1,0,1],[4838,9E+09,9E+09,9E+09,9E+09,9E+09]],[[296.85,14.1164,107.225],[0.046247,0.705593,0.705593,-0.046247],[-1,0,-1,0],[4838,9E+09,9E+09,9E+09,9E+09,9E+09]],[[296.85,-4.72739E-06,108.15],[3.09086E-08,-0.707107,-0.707107,-3.09086E-08],[-1,0,-1,0],[4838,9E+09,9E+09,9E+09,9E+09,9E+09]],[[652.53,-493.33,1047.99],[0.459259,-0.544323,-0.447932,-0.54051],[-1,0,-1,0],[4837,9E+09,9E+09,9E+09,9E+09,9E+09]],[[652.53,-493.33,1047.99],[0.459259,-0.544323,-0.447932,-0.54051],[-1,0,-2,1],[4837,9E+09,9E+09,9E+09,9E+09,9E+09]],[[652.53,-493.33,1047.99],[0.459259,-0.544323,-0.447932,-0.54051],[-1,0,-2,1],[4837,9E+09,9E+09,9E+09,9E+09,9E+09]],[[652.53,-493.33,1047.99],[0.459259,-0.544323,-0.447932,-0.54051],[-1,0,-2,1],[4837,9E+09,9E+09,9E+09,9E+09,9E+09]],[[652.53,-493.33,1047.99],[0.459259,-0.544323,-0.447932,-0.54051],[-1,0,-2,1],[4837,9E+09,9E+09,9E+09,9E+09,9E+09]],[[652.53,-493.33,1047.99],[0.459259,-0.544323,-0.447932,-0.54051],[-1,0,-2,1],[4837,9E+09,9E+09,9E+09,9E+09,9E+09]],[[652.53,-493.33,1047.99],[0.459259,-0.544323,-0.447932,-0.54051],[-1,0,-2,1],[4837,9E+09,9E+09,9E+09,9E+09,9E+09]]];
    TASK PERS robtarget robtSPHLinerFrom:=[[3794.9,108.15,88.5913],[0.5,0.5,0.5,-0.5],[-1,-1,-1,1],[1334,9E+09,9E+09,9E+09,9E+09,9E+09]];
    TASK PERS robtarget robtSPHLinerTo:=[[3794.9,108.15,-88.5913],[0.5,0.5,0.5,-0.5],[-1,-1,-1,1],[1334,9E+09,9E+09,9E+09,9E+09,9E+09]];

    !Scan platoon header results, shared for all the four scan methods
    TASK PERS pose poseSPHs{20}:=[[[0.0185547,-0.775055,0.0198339],[1,0,0,0]],[[-0.00341797,-0.529663,-0.0916748],[1,0,0,0]],[[0.012207,-0.204147,-0.0718937],[1,0,0,0]],[[-0.0161133,0.258675,0.104507],[1,0,0,0]],[[0.0166016,0.295151,0.156261],[1,0,0,0]],[[-0.0166016,0.667259,0.319176],[1,0,0,0]],[[-0.0131836,0.722885,0.481503],[1,0,0,0]],[[0.00585938,1.11372,0.896355],[1,0,0,0]],[[-0.0136719,1.26942,1.31091],[1,0,0,0]],[[0.00927734,1.46615,1.56876],[1,0,0,0]],[[0.00390625,1.28834,1.82976],[1,0,0,0]],[[-0.00341797,1.30619,2.39091],[1,0,0,0]],[[-0.0112305,1.24214,2.76328],[1,0,0,0]],[[0,0,0],[1,0,0,0]],[[0,0,0],[1,0,0,0]],[[0,0,0],[1,0,0,0]],[[0,0,0],[1,0,0,0]],[[0,0,0],[1,0,0,0]],[[0,0,0],[1,0,0,0]],[[0,0,0],[1,0,0,0]]];
    TASK PERS num numSPHLaserValues{100}:=[0,0,0,0,0,0,0,0,0,0,0,0,0,0,0,0,0,0,0,0,0,0,0,0,0,0,0,0,0,0,0,0,0,0,0,0,0,0,0,0,0,0,0,0,0,0,0,0,0,0,0,0,0,0,0,0,0,0,0,0,0,0,0,0,0,0,0,0,0,0,0,0,0,0,0,0,0,0,0,0,0,0,0,0,0,0,0,0,0,0,0,0,0,0,0,0,0,0,0,0];
    TASK PERS robtarget robtSPHPeripherys{100}:=[[[4121.12,107.375,0.0198339],[0.500025,0.49999,0.499985,-0.500001],[0,0,0,1],[1159,9E+09,9E+09,9E+09,9E+09,9E+09]],[[4121.1,107.122,10.274],[0.475432,0.523442,0.523413,-0.475406],[0,0,0,1],[1159,9E+09,9E+09,9E+09,9E+09,9E+09]],[[4121.11,105.959,20.5641],[0.449768,0.545632,0.545633,-0.449755],[0,0,0,1],[1159,9E+09,9E+09,9E+09,9E+09,9E+09]],[[4121.08,103.955,30.8208],[0.423086,0.566559,0.566566,-0.423097],[0,0,0,1],[1159,9E+09,9E+09,9E+09,9E+09,9E+09]],[[4121.12,100.57,40.67],[0.395438,0.586206,0.586201,-0.395424],[0,0,0,1],[1159,9E+09,9E+09,9E+09,9E+09,9E+09]],[[4121.08,96.5975,50.2573],[0.366812,0.604519,0.604522,-0.366823],[0,0,0,1],[1159,9E+09,9E+09,9E+09,9E+09,9E+09]],[[4121.09,91.4251,59.3842],[0.337404,0.621405,0.621421,-0.337418],[0,0,-1,1],[1159,9E+09,9E+09,9E+09,9E+09,9E+09]],[[4121.11,85.7528,68.2213],[0.307211,0.636891,0.636881,-0.307204],[0,0,-1,1],[1159,9E+09,9E+09,9E+09,9E+09,9E+09]],[[4121.09,79.066,76.4382],[0.276304,0.650842,0.650914,-0.276354],[0,0,-1,1],[1159,9E+09,9E+09,9E+09,9E+09,9E+09]],[[4121.11,71.704,83.8067],[0.244708,0.663428,0.663411,-0.244677],[0,0,-1,1],[1159,9E+09,9E+09,9E+09,9E+09,9E+09]],[[4121.1,63.3206,90.4211],[0.212624,0.674368,0.674394,-0.212631],[0,0,-1,1],[1159,9E+09,9E+09,9E+09,9E+09,9E+09]],[[4121.1,54.5618,96.5199],[0.180035,0.683793,0.683812,-0.180043],[0,1,-2,1],[1159,9E+09,9E+09,9E+09,9E+09,9E+09]],[[4121.09,45.2307,101.563],[0.147007,0.691654,0.691658,-0.147013],[0,1,-2,1],[1159,9E+09,9E+09,9E+09,9E+09,9E+09]],[[75.54,-110.49,75.53],[0.104911,-0.592891,0.59209,0.535634],[-1,-2,0,1],[3747.5,9E+09,9E+09,9E+09,9E+09,9E+09]],[[75.54,-110.49,75.53],[0.104911,-0.592891,0.59209,0.535634],[-1,0,-1,0],[3747.5,9E+09,9E+09,9E+09,9E+09,9E+09]],[[75.54,-110.49,75.53],[0.104911,-0.592891,0.59209,0.535634],[-1,0,-1,0],[3747.5,9E+09,9E+09,9E+09,9E+09,9E+09]],[[75.54,-110.49,75.53],[0.104911,-0.592891,0.59209,0.535634],[-1,0,-1,0],[3747.5,9E+09,9E+09,9E+09,9E+09,9E+09]],[[75.54,-110.49,75.53],[0.104911,-0.592891,0.59209,0.535634],[-1,0,-1,0],[3747.5,9E+09,9E+09,9E+09,9E+09,9E+09]],[[75.54,-110.49,75.53],[0.104911,-0.592891,0.59209,0.535634],[-1,0,-1,0],[3747.5,9E+09,9E+09,9E+09,9E+09,9E+09]],[[75.54,-110.49,75.53],[0.104911,-0.592891,0.59209,0.535634],[-1,0,-1,0],[3747.5,9E+09,9E+09,9E+09,9E+09,9E+09]],[[75.54,-110.49,75.53],[0.104911,-0.592891,0.59209,0.535634],[-1,0,-1,0],[3747.5,9E+09,9E+09,9E+09,9E+09,9E+09]],[[75.54,-110.49,75.53],[0.104911,-0.592891,0.59209,0.535634],[-1,0,-1,0],[3747.5,9E+09,9E+09,9E+09,9E+09,9E+09]],[[75.54,-110.49,75.53],[0.104911,-0.592891,0.59209,0.535634],[-1,0,-1,0],[3747.5,9E+09,9E+09,9E+09,9E+09,9E+09]],[[75.54,-110.49,75.53],[0.104911,-0.592891,0.59209,0.535634],[-1,0,-1,0],[3747.5,9E+09,9E+09,9E+09,9E+09,9E+09]],[[75.54,-110.49,75.53],[0.104911,-0.592891,0.59209,0.535634],[-1,0,-1,0],[3747.5,9E+09,9E+09,9E+09,9E+09,9E+09]],[[75.54,-110.49,75.53],[0.104911,-0.592891,0.59209,0.535634],[-1,0,-1,0],[3747.5,9E+09,9E+09,9E+09,9E+09,9E+09]],[[75.54,-110.49,75.53],[0.104911,-0.592891,0.59209,0.535634],[-1,0,-1,0],[3747.5,9E+09,9E+09,9E+09,9E+09,9E+09]],[[75.54,-110.49,75.53],[0.104911,-0.592891,0.59209,0.535634],[-1,0,-1,0],[3747.5,9E+09,9E+09,9E+09,9E+09,9E+09]],[[75.54,-110.49,75.53],[0.104911,-0.592891,0.59209,0.535634],[-1,0,-1,0],[3747.5,9E+09,9E+09,9E+09,9E+09,9E+09]],[[75.54,-110.49,75.53],[0.104911,-0.592891,0.59209,0.535634],[-1,0,-1,0],[3747.5,9E+09,9E+09,9E+09,9E+09,9E+09]],[[75.54,-110.49,75.53],[0.104911,-0.592891,0.59209,0.535634],[-1,0,-1,0],[3747.5,9E+09,9E+09,9E+09,9E+09,9E+09]],[[75.54,-110.49,75.53],[0.104911,-0.592891,0.59209,0.535634],[-1,0,-1,0],[3747.5,9E+09,9E+09,9E+09,9E+09,9E+09]],[[75.54,-110.49,75.53],[0.104911,-0.592891,0.59209,0.535634],[-1,0,-1,0],[3747.5,9E+09,9E+09,9E+09,9E+09,9E+09]],[[75.54,-110.49,75.53],[0.104911,-0.592891,0.59209,0.535634],[-1,0,-1,0],[3747.5,9E+09,9E+09,9E+09,9E+09,9E+09]],[[75.54,-110.49,75.53],[0.104911,-0.592891,0.59209,0.535634],[-1,0,-1,0],[3747.5,9E+09,9E+09,9E+09,9E+09,9E+09]],[[75.54,-110.49,75.53],[0.104911,-0.592891,0.59209,0.535634],[-1,0,-1,0],[3747.5,9E+09,9E+09,9E+09,9E+09,9E+09]],[[75.54,-110.49,75.53],[0.104911,-0.592891,0.59209,0.535634],[-1,0,-1,0],[3747.5,9E+09,9E+09,9E+09,9E+09,9E+09]],[[75.54,-110.49,75.53],[0.104911,-0.592891,0.59209,0.535634],[-1,0,-1,0],[3747.5,9E+09,9E+09,9E+09,9E+09,9E+09]],[[75.54,-110.49,75.53],[0.104911,-0.592891,0.59209,0.535634],[-1,0,-1,0],[3747.5,9E+09,9E+09,9E+09,9E+09,9E+09]],[[75.54,-110.49,75.53],[0.104911,-0.592891,0.59209,0.535634],[-1,0,-1,0],[3747.5,9E+09,9E+09,9E+09,9E+09,9E+09]],[[75.54,-110.49,75.53],[0.104911,-0.592891,0.59209,0.535634],[-1,0,-1,0],[3747.5,9E+09,9E+09,9E+09,9E+09,9E+09]],[[75.54,-110.49,75.53],[0.104911,-0.592891,0.59209,0.535634],[-1,0,-1,0],[3747.5,9E+09,9E+09,9E+09,9E+09,9E+09]],[[75.54,-110.49,75.53],[0.104911,-0.592891,0.59209,0.535634],[-1,0,-1,0],[3747.5,9E+09,9E+09,9E+09,9E+09,9E+09]],[[75.54,-110.49,75.53],[0.104911,-0.592891,0.59209,0.535634],[-1,0,-1,0],[3747.5,9E+09,9E+09,9E+09,9E+09,9E+09]],[[75.54,-110.49,75.53],[0.104911,-0.592891,0.59209,0.535634],[-1,0,-1,0],[3747.5,9E+09,9E+09,9E+09,9E+09,9E+09]],[[75.54,-110.49,75.53],[0.104911,-0.592891,0.59209,0.535634],[-1,0,-1,0],[3747.5,9E+09,9E+09,9E+09,9E+09,9E+09]],[[75.54,-110.49,75.53],[0.104911,-0.592891,0.59209,0.535634],[-1,0,-1,0],[3747.5,9E+09,9E+09,9E+09,9E+09,9E+09]],[[75.54,-110.49,75.53],[0.104911,-0.592891,0.59209,0.535634],[-1,0,-1,0],[3747.5,9E+09,9E+09,9E+09,9E+09,9E+09]],[[75.54,-110.49,75.53],[0.104911,-0.592891,0.59209,0.535634],[-1,0,-1,0],[3747.5,9E+09,9E+09,9E+09,9E+09,9E+09]],[[75.54,-110.49,75.53],[0.104911,-0.592891,0.59209,0.535634],[-1,0,-1,0],[3747.5,9E+09,9E+09,9E+09,9E+09,9E+09]],[[75.54,-110.49,75.53],[0.104911,-0.592891,0.59209,0.535634],[-1,0,-1,0],[3747.5,9E+09,9E+09,9E+09,9E+09,9E+09]],[[75.54,-110.49,75.53],[0.104911,-0.592891,0.59209,0.535634],[-1,0,-1,0],[3747.5,9E+09,9E+09,9E+09,9E+09,9E+09]],[[75.54,-110.49,75.53],[0.104911,-0.592891,0.59209,0.535634],[-1,0,-1,0],[3747.5,9E+09,9E+09,9E+09,9E+09,9E+09]],[[75.54,-110.49,75.53],[0.104911,-0.592891,0.59209,0.535634],[-1,0,-1,0],[3747.5,9E+09,9E+09,9E+09,9E+09,9E+09]],[[75.54,-110.49,75.53],[0.104911,-0.592891,0.59209,0.535634],[-1,0,-1,0],[3747.5,9E+09,9E+09,9E+09,9E+09,9E+09]],[[75.54,-110.49,75.53],[0.104911,-0.592891,0.59209,0.535634],[-1,0,-1,0],[3747.5,9E+09,9E+09,9E+09,9E+09,9E+09]],[[75.54,-110.49,75.53],[0.104911,-0.592891,0.59209,0.535634],[-1,0,-1,0],[3747.5,9E+09,9E+09,9E+09,9E+09,9E+09]],[[75.54,-110.49,75.53],[0.104911,-0.592891,0.59209,0.535634],[-1,0,-1,0],[3747.5,9E+09,9E+09,9E+09,9E+09,9E+09]],[[75.54,-110.49,75.53],[0.104911,-0.592891,0.59209,0.535634],[-1,0,-1,0],[3747.5,9E+09,9E+09,9E+09,9E+09,9E+09]],[[75.54,-110.49,75.53],[0.104911,-0.592891,0.59209,0.535634],[-1,0,-1,0],[3747.5,9E+09,9E+09,9E+09,9E+09,9E+09]],[[75.54,-110.49,75.53],[0.104911,-0.592891,0.59209,0.535634],[-1,0,-1,0],[3747.5,9E+09,9E+09,9E+09,9E+09,9E+09]],[[75.54,-110.49,75.53],[0.104911,-0.592891,0.59209,0.535634],[-1,0,-1,0],[3747.5,9E+09,9E+09,9E+09,9E+09,9E+09]],[[75.54,-110.49,75.53],[0.104911,-0.592891,0.59209,0.535634],[-1,0,-1,0],[3747.5,9E+09,9E+09,9E+09,9E+09,9E+09]],[[75.54,-110.49,75.53],[0.104911,-0.592891,0.59209,0.535634],[-1,0,-1,0],[3747.5,9E+09,9E+09,9E+09,9E+09,9E+09]],[[75.54,-110.49,75.53],[0.104911,-0.592891,0.59209,0.535634],[-1,0,-1,0],[3747.5,9E+09,9E+09,9E+09,9E+09,9E+09]],[[75.54,-110.49,75.53],[0.104911,-0.592891,0.59209,0.535634],[-1,0,-1,0],[3747.5,9E+09,9E+09,9E+09,9E+09,9E+09]],[[75.54,-110.49,75.53],[0.104911,-0.592891,0.59209,0.535634],[-1,0,-1,0],[3747.5,9E+09,9E+09,9E+09,9E+09,9E+09]],[[75.54,-110.49,75.53],[0.104911,-0.592891,0.59209,0.535634],[-1,0,-1,0],[3747.5,9E+09,9E+09,9E+09,9E+09,9E+09]],[[75.54,-110.49,75.53],[0.104911,-0.592891,0.59209,0.535634],[-1,0,-1,0],[3747.5,9E+09,9E+09,9E+09,9E+09,9E+09]],[[75.54,-110.49,75.53],[0.104911,-0.592891,0.59209,0.535634],[-1,0,-1,0],[3747.5,9E+09,9E+09,9E+09,9E+09,9E+09]],[[75.54,-110.49,75.53],[0.104911,-0.592891,0.59209,0.535634],[-1,0,-1,0],[3747.5,9E+09,9E+09,9E+09,9E+09,9E+09]],[[75.54,-110.49,75.53],[0.104911,-0.592891,0.59209,0.535634],[-1,0,-1,0],[3747.5,9E+09,9E+09,9E+09,9E+09,9E+09]],[[75.54,-110.49,75.53],[0.104911,-0.592891,0.59209,0.535634],[-1,0,-1,0],[3747.5,9E+09,9E+09,9E+09,9E+09,9E+09]],[[75.54,-110.49,75.53],[0.104911,-0.592891,0.59209,0.535634],[-1,0,-1,0],[3747.5,9E+09,9E+09,9E+09,9E+09,9E+09]],[[75.54,-110.49,75.53],[0.104911,-0.592891,0.59209,0.535634],[-1,0,-1,0],[3747.5,9E+09,9E+09,9E+09,9E+09,9E+09]],[[75.54,-110.49,75.53],[0.104911,-0.592891,0.59209,0.535634],[-1,0,-1,0],[3747.5,9E+09,9E+09,9E+09,9E+09,9E+09]],[[75.54,-110.49,75.53],[0.104911,-0.592891,0.59209,0.535634],[-1,0,-1,0],[3747.5,9E+09,9E+09,9E+09,9E+09,9E+09]],[[75.54,-110.49,75.53],[0.104911,-0.592891,0.59209,0.535634],[-1,0,-1,0],[3747.5,9E+09,9E+09,9E+09,9E+09,9E+09]],[[75.54,-110.49,75.53],[0.104911,-0.592891,0.59209,0.535634],[-1,0,-1,0],[3747.5,9E+09,9E+09,9E+09,9E+09,9E+09]],[[75.54,-110.49,75.53],[0.104911,-0.592891,0.59209,0.535634],[-1,0,-1,0],[3747.5,9E+09,9E+09,9E+09,9E+09,9E+09]],[[75.54,-110.49,75.53],[0.104911,-0.592891,0.59209,0.535634],[-1,0,-1,0],[3747.5,9E+09,9E+09,9E+09,9E+09,9E+09]],[[75.54,-110.49,75.53],[0.104911,-0.592891,0.59209,0.535634],[-1,0,-1,0],[3747.5,9E+09,9E+09,9E+09,9E+09,9E+09]],[[75.54,-110.49,75.53],[0.104911,-0.592891,0.59209,0.535634],[-1,0,-1,0],[3747.5,9E+09,9E+09,9E+09,9E+09,9E+09]],[[75.54,-110.49,75.53],[0.104911,-0.592891,0.59209,0.535634],[-1,0,-1,0],[3747.5,9E+09,9E+09,9E+09,9E+09,9E+09]],[[75.54,-110.49,75.53],[0.104911,-0.592891,0.59209,0.535634],[-1,0,-1,0],[3747.5,9E+09,9E+09,9E+09,9E+09,9E+09]],[[75.54,-110.49,75.53],[0.104911,-0.592891,0.59209,0.535634],[-1,0,-1,0],[3747.5,9E+09,9E+09,9E+09,9E+09,9E+09]],[[75.54,-110.49,75.53],[0.104911,-0.592891,0.59209,0.535634],[-1,0,-1,0],[3747.5,9E+09,9E+09,9E+09,9E+09,9E+09]],[[75.54,-110.49,75.53],[0.104911,-0.592891,0.59209,0.535634],[-1,0,-1,0],[3747.5,9E+09,9E+09,9E+09,9E+09,9E+09]],[[75.54,-110.49,75.53],[0.104911,-0.592891,0.59209,0.535634],[-1,0,-1,0],[3747.5,9E+09,9E+09,9E+09,9E+09,9E+09]],[[75.54,-110.49,75.53],[0.104911,-0.592891,0.59209,0.535634],[-1,0,-1,0],[3747.5,9E+09,9E+09,9E+09,9E+09,9E+09]],[[75.54,-110.49,75.53],[0.104911,-0.592891,0.59209,0.535634],[-1,0,-1,0],[3747.5,9E+09,9E+09,9E+09,9E+09,9E+09]],[[75.54,-110.49,75.53],[0.104911,-0.592891,0.59209,0.535634],[-1,0,-1,0],[3747.5,9E+09,9E+09,9E+09,9E+09,9E+09]],[[75.54,-110.49,75.53],[0.104911,-0.592891,0.59209,0.535634],[-1,0,-1,0],[3747.5,9E+09,9E+09,9E+09,9E+09,9E+09]],[[75.54,-110.49,75.53],[0.104911,-0.592891,0.59209,0.535634],[-1,0,-1,0],[3747.5,9E+09,9E+09,9E+09,9E+09,9E+09]],[[75.54,-110.49,75.53],[0.104911,-0.592891,0.59209,0.535634],[-1,0,-1,0],[3747.5,9E+09,9E+09,9E+09,9E+09,9E+09]],[[75.54,-110.49,75.53],[0.104911,-0.592891,0.59209,0.535634],[-1,0,-1,0],[3747.5,9E+09,9E+09,9E+09,9E+09,9E+09]],[[75.54,-110.49,75.53],[0.104911,-0.592891,0.59209,0.535634],[-1,0,-1,0],[3747.5,9E+09,9E+09,9E+09,9E+09,9E+09]],[[75.54,-110.49,75.53],[0.104911,-0.592891,0.59209,0.535634],[-1,0,-1,0],[3747.5,9E+09,9E+09,9E+09,9E+09,9E+09]],[[75.54,-110.49,75.53],[0.104911,-0.592891,0.59209,0.535634],[-1,0,-1,0],[3747.5,9E+09,9E+09,9E+09,9E+09,9E+09]],[[75.54,-110.49,75.53],[0.104911,-0.592891,0.59209,0.535634],[-1,0,-1,0],[3747.5,9E+09,9E+09,9E+09,9E+09,9E+09]]];
    TASK PERS pos posSPHPeripherys{100}:=[[3794.89,85.05,68.6116],[3794.89,86.6327,66.748],[3794.89,87.687,64.7089],[3794.9,72.3038,82.3319],[3794.9,74.4834,80.4222],[3794.9,75.9542,78.4286],[3794.9,78.4202,76.5584],[3794.9,80.0536,74.5451],[3794.9,81.6598,72.5306],[3794.9,83.4126,70.659],[3794.89,85.05,68.6116],[3794.89,86.6327,66.748],[3794.89,87.687,64.7089],[3794.89,89.2876,62.8192],[3794.89,90.4529,60.8162],[3794.89,91.9356,58.8769],[3794.89,92.9544,56.9193],[3794.89,93.8431,54.9808],[3794.89,94.7041,52.9993],[3794.89,96.174,51.0163],[3794.88,96.6078,49.1081],[3794.88,97.4775,47.1364],[3794.88,98.3813,45.1676],[3794.88,99.6835,42.452],[3794.89,100.27,41.2798],[3794.89,100.859,39.2845],[3794.9,101.582,37.3215],[3794.9,102.025,35.3937],[3794.9,102.753,33.4051],[3794.91,103.494,31.47],[3794.92,103.786,29.4722],[3794.92,104.207,27.5223],[3794.93,104.955,25.5668],[3794.93,105.242,23.5711],[3794.93,105.689,21.6416],[3794.92,105.398,19.6424],[3794.91,106.128,17.6712],[3794.89,106.563,15.772],[3794.88,106.856,13.7726],[3794.88,107.025,11.8457],[3794.88,107.15,9.91748],[3794.88,107.444,7.88006],[3794.87,107.166,5.95402],[3794.87,107.154,4.01375],[3794.87,106.859,2.02412],[3794.87,107.161,0.112963],[3794.87,107.166,-1.89701],[3794.88,107.016,-3.83472],[3794.88,107.166,-5.82662],[3794.89,107.019,-7.75101],[3794.89,106.865,-9.73334],[3794.89,106.563,-11.714],[3794.9,106.133,-13.641],[3794.9,105.388,-15.6283],[3794.9,105.4,-17.5522],[3794.9,105.103,-19.5513],[3794.9,104.663,-21.4851],[3794.91,104.228,-23.4668],[3794.91,103.769,-25.4156],[3794.91,103.358,-27.3991],[3794.91,102.464,-29.3372],[3794.92,102.036,-31.3149],[3794.91,101.428,-33.2104],[3794.92,100.86,-35.2208],[3794.91,99.8254,-37.1271],[3794.91,99.0964,-39.103],[3794.91,98.243,-41.0951],[3794.91,97.2104,-43.0017],[3794.9,96.4665,-45.0183],[3794.9,95.5878,-46.9843],[3794.9,94.6963,-48.8962],[3794.89,93.6819,-50.8533],[3794.89,92.5221,-52.891],[3794.89,91.1965,-54.7952],[3794.89,90.1485,-56.7162],[3794.9,88.5342,-58.7719],[3794.9,87.0889,-60.6633],[3794.91,85.4689,-62.5985],[3794.91,84.1739,-64.6154],[3794.91,82.5321,-66.606],[3794.92,81.0777,-68.354],[3794.92,79.3123,-70.4073],[3794.91,77.278,-72.3912],[3794.9,75.6686,-74.4511],[3794.9,73.1758,-76.3799],[3794.89,71.2762,-78.3072],[3794.89,69.212,-80.2458],[3794.88,66.7179,-82.1832],[3794.87,63.8071,-84.2406],[3794.87,61.469,-86.1982],[2394.11,61.4332,-88.1264],[462.953,-64.1692,-88.6888],[0,0,0],[0,0,0],[0,0,0],[0,0,0],[0,0,0],[0,0,0],[0,0,0],[0,0,0]];
    TASK PERS robtarget robtSPHPeripheryCenter:=[[3794.89,106.495,2.36952],[0.499988,0.500014,0.500009,-0.49999],[0,0,0,1],[1334,9E+09,9E+09,9E+09,9E+09,9E+09]];
    TASK PERS pose poseSPHPeripheryCenter:=[[-0.00634766,-1.65465,-0.0204563],[1,0,0,0]];

    TASK PERS jointtarget jointSPApproach:=[[-22.9735,44.092,40.4408,-40.2707,-68.9316,56.447],[4837,9E+09,9E+09,9E+09,9E+09,9E+09]];
    TASK PERS jointtarget jointSPDepart:=[[8.01002,30.801,53.756,5.52294,-56.1718,6.14333],[4837,9E+09,9E+09,9E+09,9E+09,9E+09]];

    VAR iodev iodevSPBLog;
    VAR iodev iodevSPHLog;

    TASK PERS num numSPHLLSInterval:=0.103616;
    TASK PERS num numSPHLLSScan:=90;
    TASK PERS pos posSPHLLSClosest:=[3794.88,107.444,7.88006];
    TASK PERS num numSPHLLSClosestLaseValue:=0.7004;
    TASK PERS num numSPHLLSClosestIndex:=42;
    VAR intnum intSPHLinerLaserScan;

    TASK PERS num numSPBLLSInterval:=0.1;
    TASK PERS num numSPBLLSScan:=82;
    TASK PERS pos posSPBLLSClosest:=[3250.97,38.8752,268.151];
    TASK PERS num numSPBLLSClosestLaseValue:=-0.773644;
    TASK PERS num numSPBLLSClosestIndex:=40;
    VAR intnum intSPBLinerLaserScan;

    TASK PERS speeddata speedLinearScan:=[19,500,5000,1000];

    VAR pos center;
    VAR num radius;
    VAR pos normal;
    VAR num rms;
    VAR num maxErr;
    VAR num indexWorst;

    !For Test
    TASK PERS robtarget robtBranchCenter:=[[0,0,276],[9.65967E-07,0.734915,0.678159,-1.50085E-06],[0,-1,0,0],[4837,9E+09,9E+09,9E+09,9E+09,9E+09]];
    TASK PERS robtarget robtHeaderCenter:=[[81.67,0,0],[0.675157,-0.210149,-0.675157,0.21015],[0,-1,-1,0],[4437,9E+09,9E+09,9E+09,9E+09,9E+09]];
    TASK PERS jointtarget jointBranchCenter:=[[1.52232,36.3967,-16.4912,-6.31252,34.2333,9.7168],[4837,9E+09,9E+09,9E+09,9E+09,9E+09]];
    TASK PERS jointtarget jointHeaderCenter:=[[11.9884,70.7814,-24.0764,-75.6635,62.4329,-9.61948],[4437,9E+09,9E+09,9E+09,9E+09,9E+09]];
    TASK PERS robtarget robtSTN1Aligned:=[[381.00,-38.70,119.41],[0.489644,-0.489733,-0.510175,-0.510031],[-1,0,1,1],[4838,9E+09,9E+09,9E+09,9E+09,9E+09]];
    TASK PERS jointtarget jointSTN1Aligned:=[[-0.192923,11.1632,56.797,2.35161,-31.4728,177.014],[4202,9E+09,9E+09,9E+09,9E+09,9E+09]];

    TASK PERS robtarget robtPBCenter:=[[0,0,310],[3.45176E-05,-0.720105,-0.693865,-2.60775E-05],[0,-1,0,0],[2602,9E+09,9E+09,9E+09,9E+09,9E+09]];
    TASK PERS robtarget robtPBBottom:=[[48.1,38.1,108.15],[3.09086E-08,-3.09086E-08,0.707107,-0.707107],[-1,-1,-2,1],[1967,9E+09,9E+09,9E+09,9E+09,9E+09]];
    TASK PERS robtarget robtPHCenter:=[[142.53,0,0],[0.641112,-0.298296,-0.641105,0.298295],[0,0,-2,1],[759,9E+09,9E+09,9E+09,9E+09,9E+09]];
    TASK PERS jointtarget jointPBCenter:=[[0.0298617,41.8452,-5.7915,-0.639984,17.7728,0.492516],[2602,9E+09,9E+09,9E+09,9E+09,9E+09]];
    TASK PERS jointtarget jointPBBottom:=[[-11.5611,57.2698,33.5775,-47.751,-90.5208,-91.1457],[1967,9E+09,9E+09,9E+09,9E+09,9E+09]];
    TASK PERS jointtarget jointPHCenter:=[[-17.2617,88.68,-35.5338,87.4108,65.8134,-19.3716],[3409,9E+09,9E+09,9E+09,9E+09,9E+09]];
    TASK PERS jointtarget jointPHCenter2:=[[14.3746,89.1033,-34.561,91.8377,-63.4527,-163.65],[759,9E+09,9E+09,9E+09,9E+09,9E+09]];
    TASK PERS robtarget robtPlatoonAligned:=[[2108.00,-21.16,116.06],[0.495018,-0.49502,-0.504932,-0.504932],[-1,0,-3,1],[3109,9E+09,9E+09,9E+09,9E+09,9E+09]];
    TASK PERS jointtarget jointPlatoonAligned:=[[-1.35298,49.4559,34.9342,-0.583296,-47.8646,-180.327],[3109,9E+09,9E+09,9E+09,9E+09,9E+09]];
    TASK PERS jointtarget jointPHCenterMedianLine:=[[9.05007,8.01678,48.537,4.63622,-20.9828,-171.558],[2602,9E+09,9E+09,9E+09,9E+09,9E+09]];
    TASK PERS robtarget robtPHCenterMedianLine:=[[0,133.7,0],[0.455326,0.455327,-0.540995,0.540999],[0,0,-2,1],[2602,9E+09,9E+09,9E+09,9E+09,9E+09]];
    TASK PERS jointtarget jointSHCenterMedianLine:=[[23.5615,77.3976,-15.0591,99.1075,-66.2014,-158.956],[4502,9E+09,9E+09,9E+09,9E+09,9E+09]];
    TASK PERS robtarget robtSHCenterMedianLine:=[[144.04,0,0],[0.673965,0.213937,-0.673967,-0.213939],[-1,-2,1,1],[759,9E+09,9E+09,9E+09,9E+09,9E+09]];

    TASK PERS jointtarget jointTrackHorizontal:=[[1.03407,20.8914,34.383,0.768791,-91.4422,-1.19745],[0,9E+09,9E+09,9E+09,9E+09,9E+09]];
    TASK PERS robtarget robtTrackHorizontal:=[[5217,185,1030],[0.5,0.5,0.5,-0.5],[0,0,-1,1],[0,9E+09,9E+09,9E+09,9E+09,9E+09]];

    !*****************************************************
    !For ScanV2Module
    CONST string strRobNo:="2";
    CONST string strAiLaserName:="aiLaserScan"+strRobNo;
    CONST num numTCPLaserValue:=0;

    CONST string strScanPlatoonBranchLogFileName:="ScanPlatoonBranch"+strRobNo+".csv";
    CONST string strScanPlatoonHeaderLogFileName:="ScanPlatoonHeader"+strRobNo+".csv";
    CONST string strScanSaddleBranchLogFileName:="ScanSaddleBranch"+strRobNo+".csv";
    CONST string strScanSaddleHeaderLogFileName:="ScanSaddleHeader"+strRobNo+".csv";

    TASK PERS robtarget robtSPBLLCCenter:=[[3770,38.1,293.7],[0.5,0.5,0.5,-0.5],[-1,-1,1,1],[1447,9E+09,9E+09,9E+09,9E+09,9E+09]];
    TASK PERS robtarget robtSPBLLClosestDetect:=[[3770,38.1,293.7],[0.707107,0.707107,0,0],[-1,-1,1,1],[1447,9E+09,9E+09,9E+09,9E+09,9E+09]];

    TASK PERS robtarget robtSPHLLCCenter:=[[2703.1,133.7,0],[0.5,0.5,0.5,-0.5],[0,0,1,1],[2602,9E+09,9E+09,9E+09,9E+09,9E+09]];
    TASK PERS robtarget robtSPHLLClosestDetect:=[[2703.1,133.7,0],[0.5,0.5,0.5,-0.5],[0,0,1,1],[2602,9E+09,9E+09,9E+09,9E+09,9E+09]];

    TASK PERS robtarget robtSSBLLCCenter:=[[955,-159.25,259.25],[3.09086E-08,3.09086E-08,-0.707107,-0.707107],[-1,-1,1,1],[4262,9E+09,9E+09,9E+09,9E+09,9E+09]];
    TASK PERS robtarget robtSSBLLClosestDetect:=[[955,-38.1,268.15],[3.09086E-08,3.09086E-08,-0.707107,-0.707107],[-1,-1,1,1],[4262,9E+09,9E+09,9E+09,9E+09,9E+09]];

    TASK PERS robtarget robtSSHLLCCenter:=[[462.15,-108.15,0],[0.5,-0.5,-0.5,-0.5],[0,0,1,1],[4837,9E+9,9E+9,9E+9,9E+9,9E+9]];
    TASK PERS robtarget robtSSHLLClosestDetect:=[[462.15,-108.15,0],[0.5,-0.5,-0.5,-0.5],[0,0,1,1],[4837,9E+9,9E+9,9E+9,9E+9,9E+9]];
    !*****************************************************

ENDMODULE
